REGION Network 47: Call CM Master Virtual Axis (LER_Interlock Summary)
   RUNG wire#powerrail
      #instCmMasterAxisControlInterlockSummary(enableManualCmds := wire#w1, interlockSource := "Unit1.Em3.ControlNodes".cm.Interlock.masterVirtualAxis.source, moduleInterface := "Unit1.Em3.HmiInterface".cmMasterVirtualAxis, controlNode := "Unit1.Em3.ControlNodes".cmMasterVirtualAxis, interlockcGeneral => "Unit1.Em3.ControlNodes".cm.Interlock.masterVirtualAxis.permit.general)
   END_RUNG
   RUNG wire#powerrail
      I_Contact( #statUnitStatus.mode.production )
      Contact( "Unit1.Em3.HmiInterface".webGuid.sequence.monitoring.inStepIdle )
   END_RUNG wire#w1
   // the same network as SCL:
   #instCmMasterAxisControlInterlockSummary(enableManualCmds := NOT #statUnitStatus.mode.production AND "Unit1.Em3.HmiInterface".webGuid.sequence.monitoring.inStepIdle,   // "LER_AxisControl_InterlockSummary"
                           interlockSource := "Unit1.Em3.ControlNodes".cm.Interlock.masterVirtualAxis.source,
                           moduleInterface := "Unit1.Em3.HmiInterface".cmMasterVirtualAxis,
                           controlNode := "Unit1.Em3.ControlNodes".cmMasterVirtualAxis,
                           interlockcGeneral => "Unit1.Em3.ControlNodes".cm.Interlock.masterVirtualAxis.permit.general);
END_REGION

REGION Network 48: Call CM Master Virtual Axis (LBC_AxisControl)
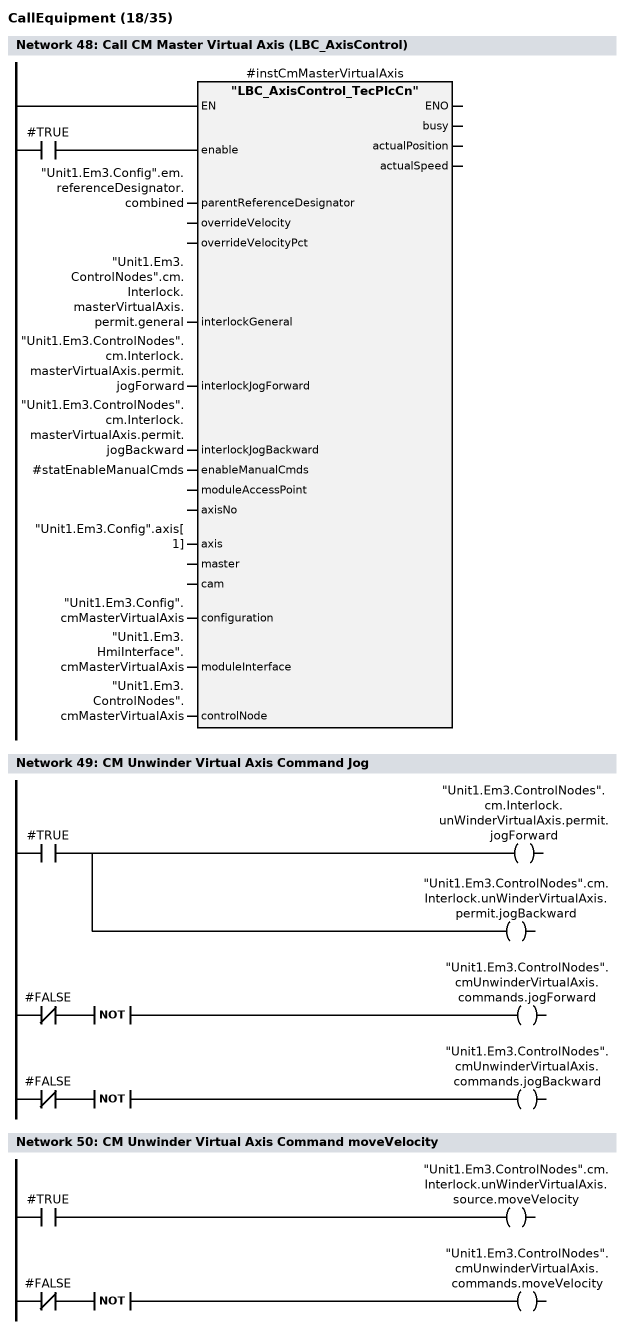
   RUNG wire#powerrail
      #instCmMasterVirtualAxis(enable := wire#w1, parentReferenceDesignator := "Unit1.Em3.Config".em.referenceDesignator.combined, overrideVelocity :=, overrideVelocityPct :=, interlockGeneral := "Unit1.Em3.ControlNodes".cm.Interlock.masterVirtualAxis.permit.general, interlockJogForward := "Unit1.Em3.ControlNodes".cm.Interlock.masterVirtualAxis.permit.jogForward, interlockJogBackward := "Unit1.Em3.ControlNodes".cm.Interlock.masterVirtualAxis.permit.jogBackward, enableManualCmds := #statEnableManualCmds, moduleAccessPoint :=, axisNo :=, axis := "Unit1.Em3.Config".axis[1], master :=, cam :=, configuration := "Unit1.Em3.Config".cmMasterVirtualAxis, moduleInterface := "Unit1.Em3.HmiInterface".cmMasterVirtualAxis, controlNode := "Unit1.Em3.ControlNodes".cmMasterVirtualAxis, busy =>, actualPosition =>, actualSpeed =>)
   END_RUNG
   RUNG wire#powerrail
      Contact( #TRUE )
   END_RUNG wire#w1
   // the same network as SCL:
   #instCmMasterVirtualAxis(enable := #TRUE,   // "LBC_AxisControl_TecPlcCn"
                           parentReferenceDesignator := "Unit1.Em3.Config".em.referenceDesignator.combined,
                           interlockGeneral := "Unit1.Em3.ControlNodes".cm.Interlock.masterVirtualAxis.permit.general,
                           interlockJogForward := "Unit1.Em3.ControlNodes".cm.Interlock.masterVirtualAxis.permit.jogForward,
                           interlockJogBackward := "Unit1.Em3.ControlNodes".cm.Interlock.masterVirtualAxis.permit.jogBackward,
                           enableManualCmds := #statEnableManualCmds,
                           axis := "Unit1.Em3.Config".axis[1],
                           configuration := "Unit1.Em3.Config".cmMasterVirtualAxis,
                           moduleInterface := "Unit1.Em3.HmiInterface".cmMasterVirtualAxis,
                           controlNode := "Unit1.Em3.ControlNodes".cmMasterVirtualAxis);
END_REGION

REGION Network 49: CM Unwinder Virtual Axis Command Jog
   RUNG wire#powerrail
      Contact( #TRUE )
      wire#w1
      Coil( "Unit1.Em3.ControlNodes".cm.Interlock.unWinderVirtualAxis.permit.jogForward )
   END_RUNG
   RUNG wire#w1
      Coil( "Unit1.Em3.ControlNodes".cm.Interlock.unWinderVirtualAxis.permit.jogBackward )
   END_RUNG
   RUNG wire#powerrail
      I_Contact( #FALSE )
      Not()
      Coil( "Unit1.Em3.ControlNodes".cmUnwinderVirtualAxis.commands.jogForward )
   END_RUNG
   RUNG wire#powerrail
      I_Contact( #FALSE )
      Not()
      Coil( "Unit1.Em3.ControlNodes".cmUnwinderVirtualAxis.commands.jogBackward )
   END_RUNG
   // the same network as SCL:
   "Unit1.Em3.ControlNodes".cm.Interlock.unWinderVirtualAxis.permit.jogForward := #TRUE;
   "Unit1.Em3.ControlNodes".cm.Interlock.unWinderVirtualAxis.permit.jogBackward := #TRUE;
   "Unit1.Em3.ControlNodes".cmUnwinderVirtualAxis.commands.jogForward := NOT (NOT #FALSE);
   "Unit1.Em3.ControlNodes".cmUnwinderVirtualAxis.commands.jogBackward := NOT (NOT #FALSE);
END_REGION

REGION Network 50: CM Unwinder Virtual Axis Command moveVelocity
   RUNG wire#powerrail
      Contact( #TRUE )
      Coil( "Unit1.Em3.ControlNodes".cm.Interlock.unWinderVirtualAxis.source.moveVelocity )
   END_RUNG
   RUNG wire#powerrail
      I_Contact( #FALSE )
      Not()
      Coil( "Unit1.Em3.ControlNodes".cmUnwinderVirtualAxis.commands.moveVelocity )
   END_RUNG
   // the same network as SCL:
   "Unit1.Em3.ControlNodes".cm.Interlock.unWinderVirtualAxis.source.moveVelocity := #TRUE;
   "Unit1.Em3.ControlNodes".cmUnwinderVirtualAxis.commands.moveVelocity := NOT (NOT #FALSE);
END_REGION

REGION Network 51: CM Unwinder Virtual Axis Command stop
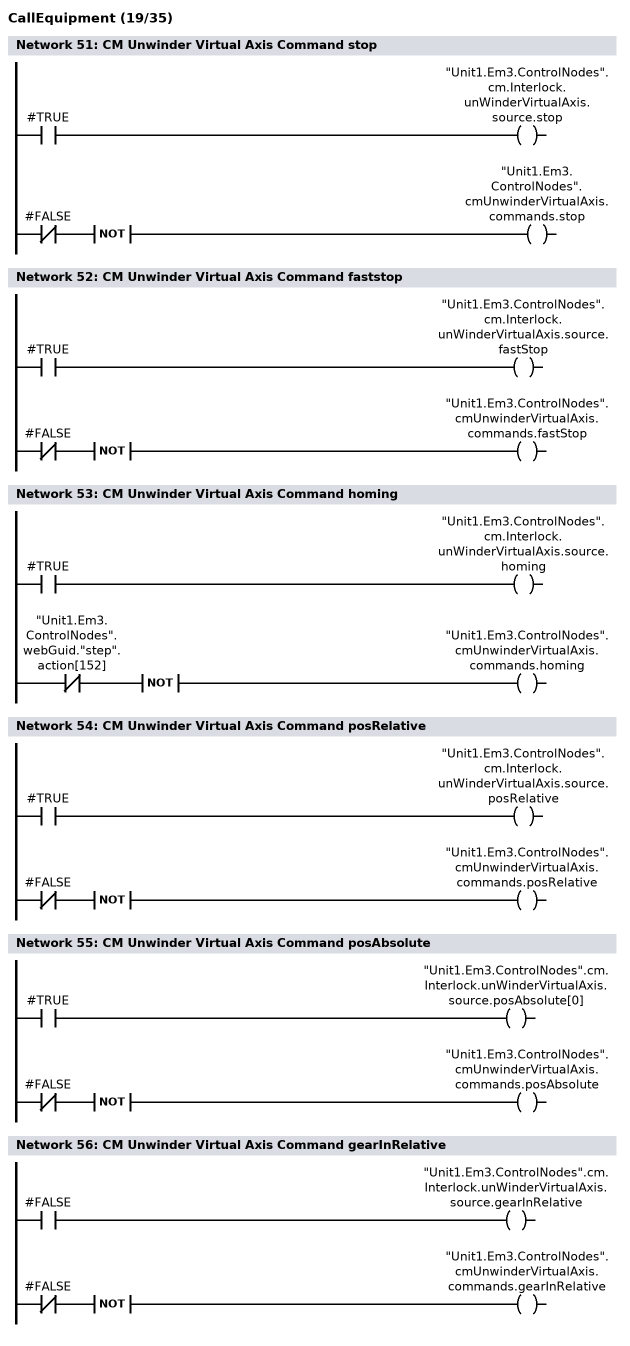
   RUNG wire#powerrail
      Contact( #TRUE )
      Coil( "Unit1.Em3.ControlNodes".cm.Interlock.unWinderVirtualAxis.source.stop )
   END_RUNG
   RUNG wire#powerrail
      I_Contact( #FALSE )
      Not()
      Coil( "Unit1.Em3.ControlNodes".cmUnwinderVirtualAxis.commands.stop )
   END_RUNG
   // the same network as SCL:
   "Unit1.Em3.ControlNodes".cm.Interlock.unWinderVirtualAxis.source.stop := #TRUE;
   "Unit1.Em3.ControlNodes".cmUnwinderVirtualAxis.commands.stop := NOT (NOT #FALSE);
END_REGION

REGION Network 52: CM Unwinder Virtual Axis Command faststop
   RUNG wire#powerrail
      Contact( #TRUE )
      Coil( "Unit1.Em3.ControlNodes".cm.Interlock.unWinderVirtualAxis.source.fastStop )
   END_RUNG
   RUNG wire#powerrail
      I_Contact( #FALSE )
      Not()
      Coil( "Unit1.Em3.ControlNodes".cmUnwinderVirtualAxis.commands.fastStop )
   END_RUNG
   // the same network as SCL:
   "Unit1.Em3.ControlNodes".cm.Interlock.unWinderVirtualAxis.source.fastStop := #TRUE;
   "Unit1.Em3.ControlNodes".cmUnwinderVirtualAxis.commands.fastStop := NOT (NOT #FALSE);
END_REGION

REGION Network 53: CM Unwinder Virtual Axis Command homing
   RUNG wire#powerrail
      Contact( #TRUE )
      Coil( "Unit1.Em3.ControlNodes".cm.Interlock.unWinderVirtualAxis.source.homing )
   END_RUNG
   RUNG wire#powerrail
      I_Contact( "Unit1.Em3.ControlNodes".webGuid."step".action[152] )
      Not()
      Coil( "Unit1.Em3.ControlNodes".cmUnwinderVirtualAxis.commands.homing )
   END_RUNG
   // the same network as SCL:
   "Unit1.Em3.ControlNodes".cm.Interlock.unWinderVirtualAxis.source.homing := #TRUE;
   "Unit1.Em3.ControlNodes".cmUnwinderVirtualAxis.commands.homing := NOT (NOT "Unit1.Em3.ControlNodes".webGuid."step".action[152]);
END_REGION

REGION Network 54: CM Unwinder Virtual Axis Command posRelative
   RUNG wire#powerrail
      Contact( #TRUE )
      Coil( "Unit1.Em3.ControlNodes".cm.Interlock.unWinderVirtualAxis.source.posRelative )
   END_RUNG
   RUNG wire#powerrail
      I_Contact( #FALSE )
      Not()
      Coil( "Unit1.Em3.ControlNodes".cmUnwinderVirtualAxis.commands.posRelative )
   END_RUNG
   // the same network as SCL:
   "Unit1.Em3.ControlNodes".cm.Interlock.unWinderVirtualAxis.source.posRelative := #TRUE;
   "Unit1.Em3.ControlNodes".cmUnwinderVirtualAxis.commands.posRelative := NOT (NOT #FALSE);
END_REGION

REGION Network 55: CM Unwinder Virtual Axis Command posAbsolute
   RUNG wire#powerrail
      Contact( #TRUE )
      Coil( "Unit1.Em3.ControlNodes".cm.Interlock.unWinderVirtualAxis.source.posAbsolute[0] )
   END_RUNG
   RUNG wire#powerrail
      I_Contact( #FALSE )
      Not()
      Coil( "Unit1.Em3.ControlNodes".cmUnwinderVirtualAxis.commands.posAbsolute )
   END_RUNG
   // the same network as SCL:
   "Unit1.Em3.ControlNodes".cm.Interlock.unWinderVirtualAxis.source.posAbsolute[0] := #TRUE;
   "Unit1.Em3.ControlNodes".cmUnwinderVirtualAxis.commands.posAbsolute := NOT (NOT #FALSE);
END_REGION

REGION Network 56: CM Unwinder Virtual Axis Command gearInRelative
   RUNG wire#powerrail
      Contact( #FALSE )
      Coil( "Unit1.Em3.ControlNodes".cm.Interlock.unWinderVirtualAxis.source.gearInRelative )
   END_RUNG
   RUNG wire#powerrail
      I_Contact( #FALSE )
      Not()
      Coil( "Unit1.Em3.ControlNodes".cmUnwinderVirtualAxis.commands.gearInRelative )
   END_RUNG
   // the same network as SCL:
   "Unit1.Em3.ControlNodes".cm.Interlock.unWinderVirtualAxis.source.gearInRelative := #FALSE;
   "Unit1.Em3.ControlNodes".cmUnwinderVirtualAxis.commands.gearInRelative := NOT (NOT #FALSE);
END_REGION

REGION Network 57: CM Unwinder Virtual Axis Command gearInAbsolute
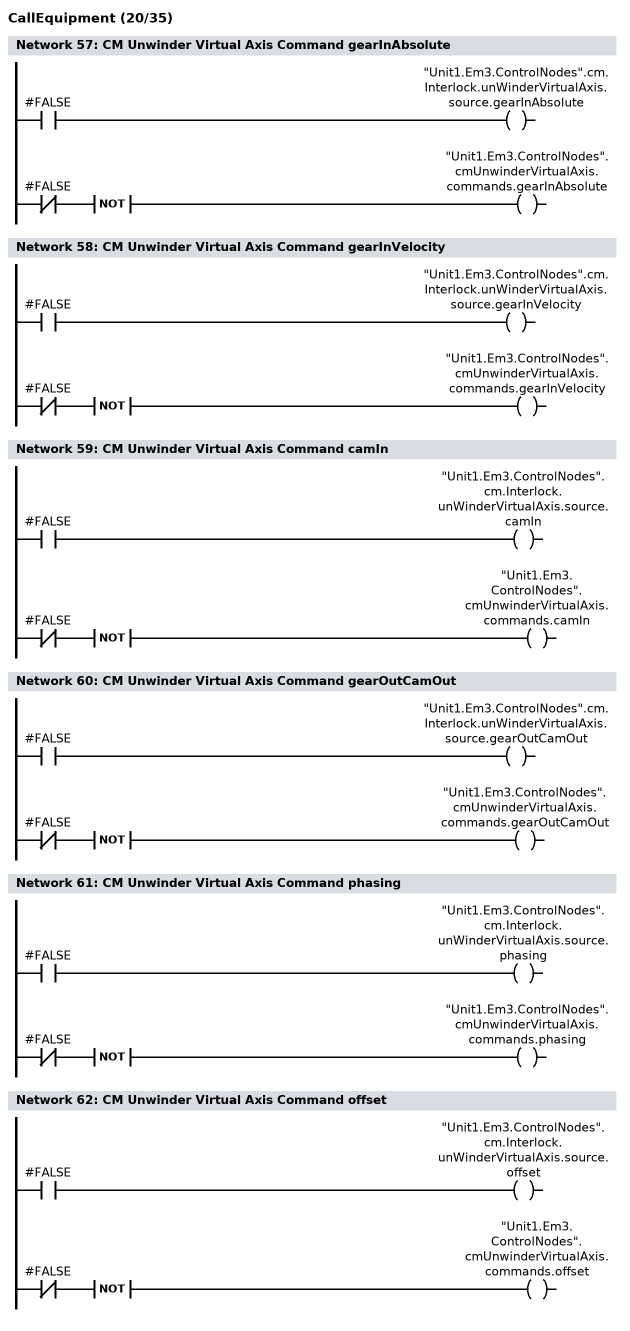
   RUNG wire#powerrail
      Contact( #FALSE )
      Coil( "Unit1.Em3.ControlNodes".cm.Interlock.unWinderVirtualAxis.source.gearInAbsolute )
   END_RUNG
   RUNG wire#powerrail
      I_Contact( #FALSE )
      Not()
      Coil( "Unit1.Em3.ControlNodes".cmUnwinderVirtualAxis.commands.gearInAbsolute )
   END_RUNG
   // the same network as SCL:
   "Unit1.Em3.ControlNodes".cm.Interlock.unWinderVirtualAxis.source.gearInAbsolute := #FALSE;
   "Unit1.Em3.ControlNodes".cmUnwinderVirtualAxis.commands.gearInAbsolute := NOT (NOT #FALSE);
END_REGION

REGION Network 58: CM Unwinder Virtual Axis Command gearInVelocity
   RUNG wire#powerrail
      Contact( #FALSE )
      Coil( "Unit1.Em3.ControlNodes".cm.Interlock.unWinderVirtualAxis.source.gearInVelocity )
   END_RUNG
   RUNG wire#powerrail
      I_Contact( #FALSE )
      Not()
      Coil( "Unit1.Em3.ControlNodes".cmUnwinderVirtualAxis.commands.gearInVelocity )
   END_RUNG
   // the same network as SCL:
   "Unit1.Em3.ControlNodes".cm.Interlock.unWinderVirtualAxis.source.gearInVelocity := #FALSE;
   "Unit1.Em3.ControlNodes".cmUnwinderVirtualAxis.commands.gearInVelocity := NOT (NOT #FALSE);
END_REGION

REGION Network 59: CM Unwinder Virtual Axis Command camIn
   RUNG wire#powerrail
      Contact( #FALSE )
      Coil( "Unit1.Em3.ControlNodes".cm.Interlock.unWinderVirtualAxis.source.camIn )
   END_RUNG
   RUNG wire#powerrail
      I_Contact( #FALSE )
      Not()
      Coil( "Unit1.Em3.ControlNodes".cmUnwinderVirtualAxis.commands.camIn )
   END_RUNG
   // the same network as SCL:
   "Unit1.Em3.ControlNodes".cm.Interlock.unWinderVirtualAxis.source.camIn := #FALSE;
   "Unit1.Em3.ControlNodes".cmUnwinderVirtualAxis.commands.camIn := NOT (NOT #FALSE);
END_REGION

REGION Network 60: CM Unwinder Virtual Axis Command gearOutCamOut
   RUNG wire#powerrail
      Contact( #FALSE )
      Coil( "Unit1.Em3.ControlNodes".cm.Interlock.unWinderVirtualAxis.source.gearOutCamOut )
   END_RUNG
   RUNG wire#powerrail
      I_Contact( #FALSE )
      Not()
      Coil( "Unit1.Em3.ControlNodes".cmUnwinderVirtualAxis.commands.gearOutCamOut )
   END_RUNG
   // the same network as SCL:
   "Unit1.Em3.ControlNodes".cm.Interlock.unWinderVirtualAxis.source.gearOutCamOut := #FALSE;
   "Unit1.Em3.ControlNodes".cmUnwinderVirtualAxis.commands.gearOutCamOut := NOT (NOT #FALSE);
END_REGION

REGION Network 61: CM Unwinder Virtual Axis Command phasing
   RUNG wire#powerrail
      Contact( #FALSE )
      Coil( "Unit1.Em3.ControlNodes".cm.Interlock.unWinderVirtualAxis.source.phasing )
   END_RUNG
   RUNG wire#powerrail
      I_Contact( #FALSE )
      Not()
      Coil( "Unit1.Em3.ControlNodes".cmUnwinderVirtualAxis.commands.phasing )
   END_RUNG
   // the same network as SCL:
   "Unit1.Em3.ControlNodes".cm.Interlock.unWinderVirtualAxis.source.phasing := #FALSE;
   "Unit1.Em3.ControlNodes".cmUnwinderVirtualAxis.commands.phasing := NOT (NOT #FALSE);
END_REGION

REGION Network 62: CM Unwinder Virtual Axis Command offset
   RUNG wire#powerrail
      Contact( #FALSE )
      Coil( "Unit1.Em3.ControlNodes".cm.Interlock.unWinderVirtualAxis.source.offset )
   END_RUNG
   RUNG wire#powerrail
      I_Contact( #FALSE )
      Not()
      Coil( "Unit1.Em3.ControlNodes".cmUnwinderVirtualAxis.commands.offset )
   END_RUNG
   // the same network as SCL:
   "Unit1.Em3.ControlNodes".cm.Interlock.unWinderVirtualAxis.source.offset := #FALSE;
   "Unit1.Em3.ControlNodes".cmUnwinderVirtualAxis.commands.offset := NOT (NOT #FALSE);
END_REGION

REGION Network 63: Call CM Unwinder Virtual Axis (LER_Interlock Summary)
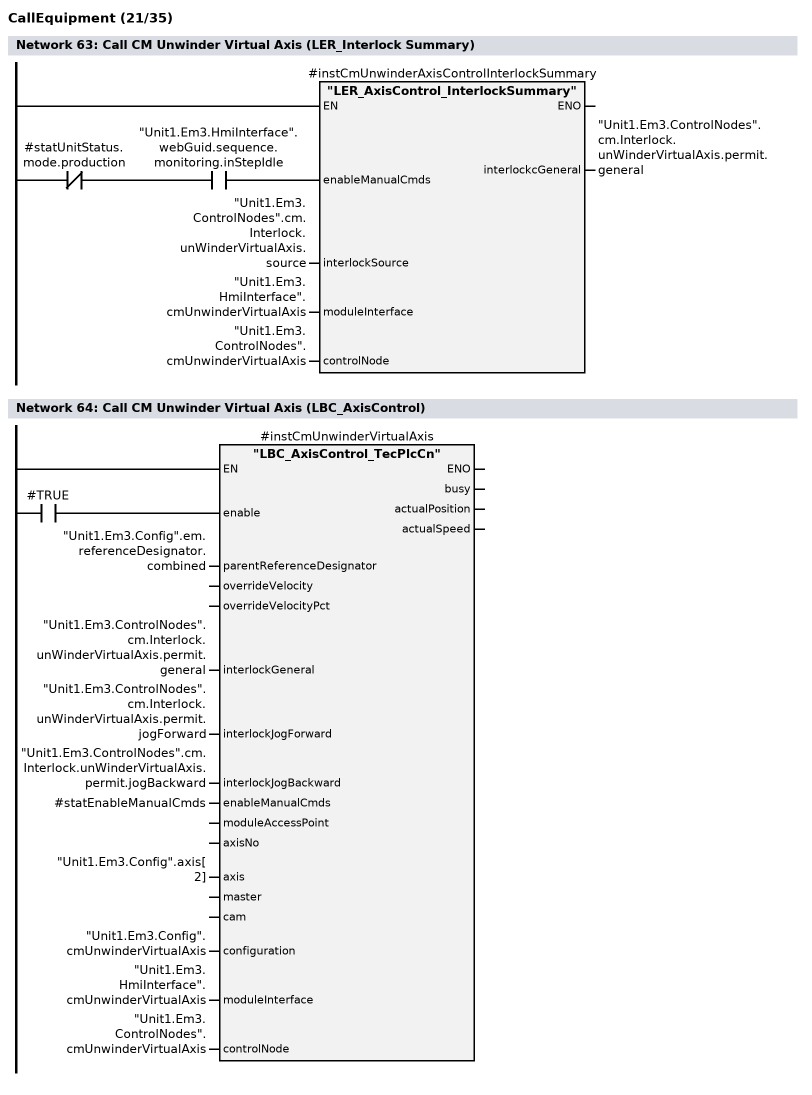
   RUNG wire#powerrail
      #instCmUnwinderAxisControlInterlockSummary(enableManualCmds := wire#w1, interlockSource := "Unit1.Em3.ControlNodes".cm.Interlock.unWinderVirtualAxis.source, moduleInterface := "Unit1.Em3.HmiInterface".cmUnwinderVirtualAxis, controlNode := "Unit1.Em3.ControlNodes".cmUnwinderVirtualAxis, interlockcGeneral => "Unit1.Em3.ControlNodes".cm.Interlock.unWinderVirtualAxis.permit.general)
   END_RUNG
   RUNG wire#powerrail
      I_Contact( #statUnitStatus.mode.production )
      Contact( "Unit1.Em3.HmiInterface".webGuid.sequence.monitoring.inStepIdle )
   END_RUNG wire#w1
   // the same network as SCL:
   #instCmUnwinderAxisControlInterlockSummary(enableManualCmds := NOT #statUnitStatus.mode.production AND "Unit1.Em3.HmiInterface".webGuid.sequence.monitoring.inStepIdle,   // "LER_AxisControl_InterlockSummary"
                           interlockSource := "Unit1.Em3.ControlNodes".cm.Interlock.unWinderVirtualAxis.source,
                           moduleInterface := "Unit1.Em3.HmiInterface".cmUnwinderVirtualAxis,
                           controlNode := "Unit1.Em3.ControlNodes".cmUnwinderVirtualAxis,
                           interlockcGeneral => "Unit1.Em3.ControlNodes".cm.Interlock.unWinderVirtualAxis.permit.general);
END_REGION

REGION Network 64: Call CM Unwinder Virtual Axis (LBC_AxisControl)
   RUNG wire#powerrail
      #instCmUnwinderVirtualAxis(enable := wire#w1, parentReferenceDesignator := "Unit1.Em3.Config".em.referenceDesignator.combined, overrideVelocity :=, overrideVelocityPct :=, interlockGeneral := "Unit1.Em3.ControlNodes".cm.Interlock.unWinderVirtualAxis.permit.general, interlockJogForward := "Unit1.Em3.ControlNodes".cm.Interlock.unWinderVirtualAxis.permit.jogForward, interlockJogBackward := "Unit1.Em3.ControlNodes".cm.Interlock.unWinderVirtualAxis.permit.jogBackward, enableManualCmds := #statEnableManualCmds, moduleAccessPoint :=, axisNo :=, axis := "Unit1.Em3.Config".axis[2], master :=, cam :=, configuration := "Unit1.Em3.Config".cmUnwinderVirtualAxis, moduleInterface := "Unit1.Em3.HmiInterface".cmUnwinderVirtualAxis, controlNode := "Unit1.Em3.ControlNodes".cmUnwinderVirtualAxis, busy =>, actualPosition =>, actualSpeed =>)
   END_RUNG
   RUNG wire#powerrail
      Contact( #TRUE )
   END_RUNG wire#w1
   // the same network as SCL:
   #instCmUnwinderVirtualAxis(enable := #TRUE,   // "LBC_AxisControl_TecPlcCn"
                           parentReferenceDesignator := "Unit1.Em3.Config".em.referenceDesignator.combined,
                           interlockGeneral := "Unit1.Em3.ControlNodes".cm.Interlock.unWinderVirtualAxis.permit.general,
                           interlockJogForward := "Unit1.Em3.ControlNodes".cm.Interlock.unWinderVirtualAxis.permit.jogForward,
                           interlockJogBackward := "Unit1.Em3.ControlNodes".cm.Interlock.unWinderVirtualAxis.permit.jogBackward,
                           enableManualCmds := #statEnableManualCmds,
                           axis := "Unit1.Em3.Config".axis[2],
                           configuration := "Unit1.Em3.Config".cmUnwinderVirtualAxis,
                           moduleInterface := "Unit1.Em3.HmiInterface".cmUnwinderVirtualAxis,
                           controlNode := "Unit1.Em3.ControlNodes".cmUnwinderVirtualAxis);
END_REGION

REGION Network 65: ******************** Control Modules (TwoWayActuator) ********************
   // Call control modules that are actuators after the em logic (jobs and sequence), so that the latest commands are applied to the actuators.
END_REGION

REGION Network 66: Reset CMS
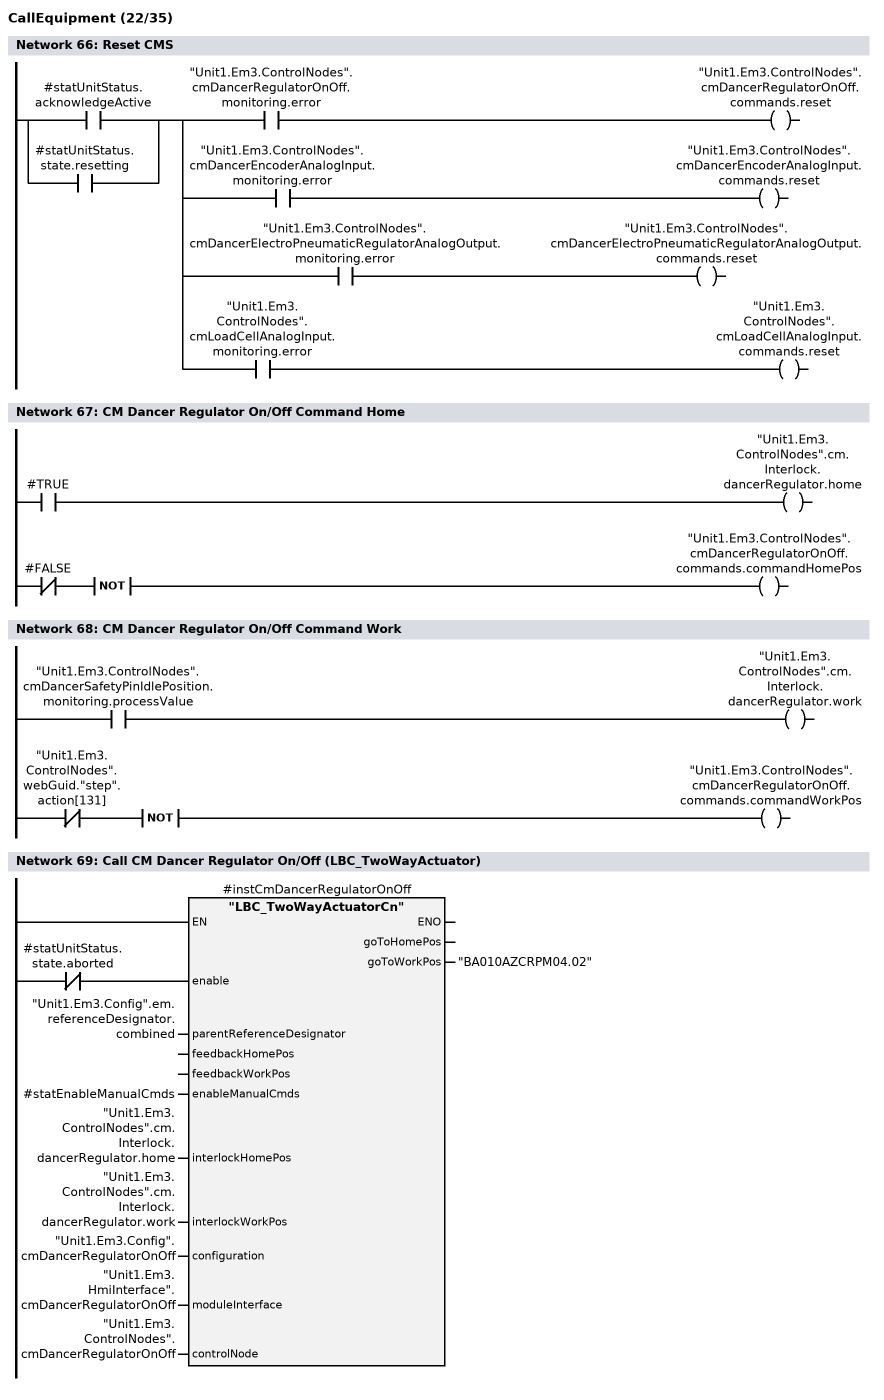
   RUNG wire#powerrail
      Contact( #statUnitStatus.acknowledgeActive )
      wire#w1
      Contact( "Unit1.Em3.ControlNodes".cmDancerRegulatorOnOff.monitoring.error )
      Coil( "Unit1.Em3.ControlNodes".cmDancerRegulatorOnOff.commands.reset )
   END_RUNG
   RUNG wire#powerrail
      Contact( #statUnitStatus.state.resetting )
   END_RUNG wire#w1
   RUNG wire#w1
      Contact( "Unit1.Em3.ControlNodes".cmDancerEncoderAnalogInput.monitoring.error )
      Coil( "Unit1.Em3.ControlNodes".cmDancerEncoderAnalogInput.commands.reset )
   END_RUNG
   RUNG wire#w1
      Contact( "Unit1.Em3.ControlNodes".cmDancerElectroPneumaticRegulatorAnalogOutput.monitoring.error )
      Coil( "Unit1.Em3.ControlNodes".cmDancerElectroPneumaticRegulatorAnalogOutput.commands.reset )
   END_RUNG
   RUNG wire#w1
      Contact( "Unit1.Em3.ControlNodes".cmLoadCellAnalogInput.monitoring.error )
      Coil( "Unit1.Em3.ControlNodes".cmLoadCellAnalogInput.commands.reset )
   END_RUNG
   // the same network as SCL:
   #_w1 := #statUnitStatus.acknowledgeActive OR #statUnitStatus.state.resetting;
   "Unit1.Em3.ControlNodes".cmDancerRegulatorOnOff.commands.reset := #_w1 AND "Unit1.Em3.ControlNodes".cmDancerRegulatorOnOff.monitoring.error;
   "Unit1.Em3.ControlNodes".cmDancerEncoderAnalogInput.commands.reset := #_w1 AND "Unit1.Em3.ControlNodes".cmDancerEncoderAnalogInput.monitoring.error;
   "Unit1.Em3.ControlNodes".cmDancerElectroPneumaticRegulatorAnalogOutput.commands.reset := #_w1 AND "Unit1.Em3.ControlNodes".cmDancerElectroPneumaticRegulatorAnalogOutput.monitoring.error;
   "Unit1.Em3.ControlNodes".cmLoadCellAnalogInput.commands.reset := #_w1 AND "Unit1.Em3.ControlNodes".cmLoadCellAnalogInput.monitoring.error;
END_REGION

REGION Network 67: CM Dancer Regulator On/Off Command Home
   RUNG wire#powerrail
      Contact( #TRUE )
      Coil( "Unit1.Em3.ControlNodes".cm.Interlock.dancerRegulator.home )
   END_RUNG
   RUNG wire#powerrail
      I_Contact( #FALSE )
      Not()
      Coil( "Unit1.Em3.ControlNodes".cmDancerRegulatorOnOff.commands.commandHomePos )
   END_RUNG
   // the same network as SCL:
   "Unit1.Em3.ControlNodes".cm.Interlock.dancerRegulator.home := #TRUE;
   "Unit1.Em3.ControlNodes".cmDancerRegulatorOnOff.commands.commandHomePos := NOT (NOT #FALSE);
END_REGION

REGION Network 68: CM Dancer Regulator On/Off Command Work
   RUNG wire#powerrail
      Contact( "Unit1.Em3.ControlNodes".cmDancerSafetyPinIdlePosition.monitoring.processValue )
      Coil( "Unit1.Em3.ControlNodes".cm.Interlock.dancerRegulator.work )
   END_RUNG
   RUNG wire#powerrail
      I_Contact( "Unit1.Em3.ControlNodes".webGuid."step".action[131] )
      Not()
      Coil( "Unit1.Em3.ControlNodes".cmDancerRegulatorOnOff.commands.commandWorkPos )
   END_RUNG
   // the same network as SCL:
   "Unit1.Em3.ControlNodes".cm.Interlock.dancerRegulator.work := "Unit1.Em3.ControlNodes".cmDancerSafetyPinIdlePosition.monitoring.processValue;
   "Unit1.Em3.ControlNodes".cmDancerRegulatorOnOff.commands.commandWorkPos := NOT (NOT "Unit1.Em3.ControlNodes".webGuid."step".action[131]);
END_REGION

REGION Network 69: Call CM Dancer Regulator On/Off (LBC_TwoWayActuator)
   RUNG wire#powerrail
      #instCmDancerRegulatorOnOff(enable := wire#w1, parentReferenceDesignator := "Unit1.Em3.Config".em.referenceDesignator.combined, feedbackHomePos :=, feedbackWorkPos :=, enableManualCmds := #statEnableManualCmds, interlockHomePos := "Unit1.Em3.ControlNodes".cm.Interlock.dancerRegulator.home, interlockWorkPos := "Unit1.Em3.ControlNodes".cm.Interlock.dancerRegulator.work, configuration := "Unit1.Em3.Config".cmDancerRegulatorOnOff, moduleInterface := "Unit1.Em3.HmiInterface".cmDancerRegulatorOnOff, controlNode := "Unit1.Em3.ControlNodes".cmDancerRegulatorOnOff, goToHomePos =>, goToWorkPos => "BA010AZCRPM04.02")
   END_RUNG
   RUNG wire#powerrail
      I_Contact( #statUnitStatus.state.aborted )
   END_RUNG wire#w1
   // the same network as SCL:
   #instCmDancerRegulatorOnOff(enable := NOT #statUnitStatus.state.aborted,   // "LBC_TwoWayActuatorCn"
                           parentReferenceDesignator := "Unit1.Em3.Config".em.referenceDesignator.combined,
                           enableManualCmds := #statEnableManualCmds,
                           interlockHomePos := "Unit1.Em3.ControlNodes".cm.Interlock.dancerRegulator.home,
                           interlockWorkPos := "Unit1.Em3.ControlNodes".cm.Interlock.dancerRegulator.work,
                           configuration := "Unit1.Em3.Config".cmDancerRegulatorOnOff,
                           moduleInterface := "Unit1.Em3.HmiInterface".cmDancerRegulatorOnOff,
                           controlNode := "Unit1.Em3.ControlNodes".cmDancerRegulatorOnOff,
                           goToWorkPos => "BA010AZCRPM04.02");
END_REGION

REGION Network 70: ******************** Control Modules (Accessories) ********************
   // Call control modules that are actuators after the em logic (jobs and sequence), so that the latest commands are applied to the actuators.
END_REGION

REGION Network 71: Reset CMS
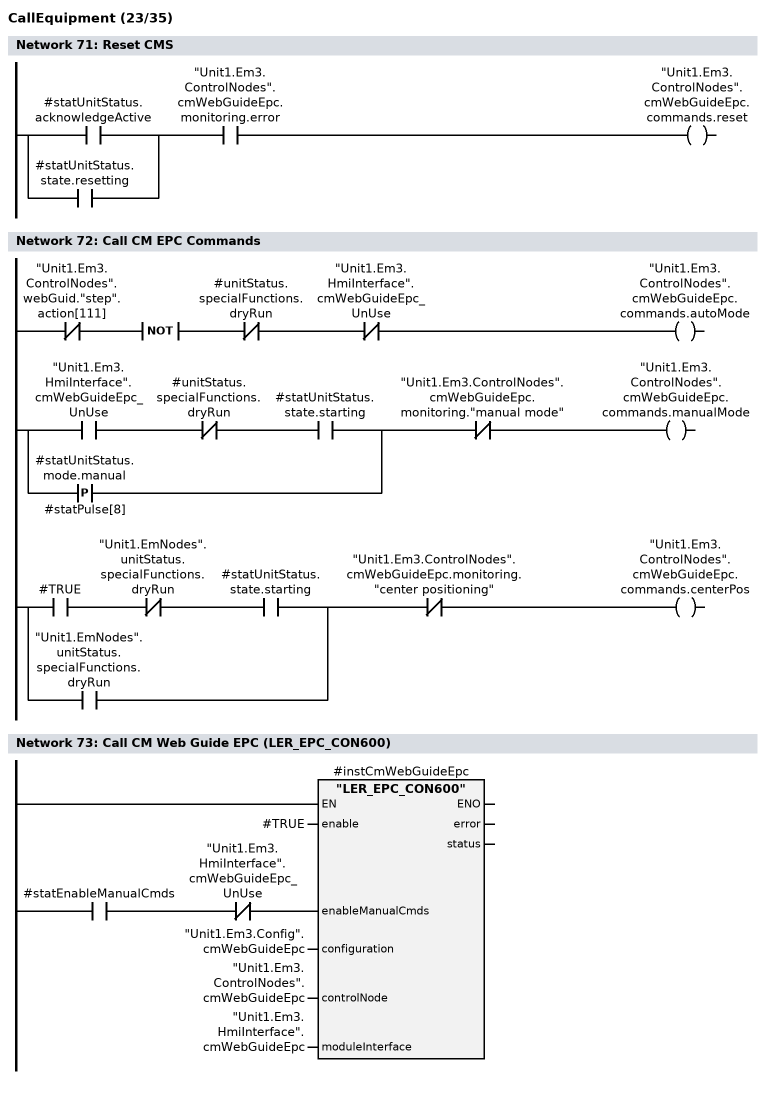
   RUNG wire#powerrail
      Contact( #statUnitStatus.acknowledgeActive )
      wire#w1
      Contact( "Unit1.Em3.ControlNodes".cmWebGuideEpc.monitoring.error )
      Coil( "Unit1.Em3.ControlNodes".cmWebGuideEpc.commands.reset )
   END_RUNG
   RUNG wire#powerrail
      Contact( #statUnitStatus.state.resetting )
   END_RUNG wire#w1
   // the same network as SCL:
   "Unit1.Em3.ControlNodes".cmWebGuideEpc.commands.reset := (#statUnitStatus.acknowledgeActive OR #statUnitStatus.state.resetting) AND "Unit1.Em3.ControlNodes".cmWebGuideEpc.monitoring.error;
END_REGION

REGION Network 72: Call CM EPC Commands
   RUNG wire#powerrail
      I_Contact( "Unit1.Em3.ControlNodes".webGuid."step".action[111] )
      Not()
      I_Contact( #unitStatus.specialFunctions.dryRun )
      I_Contact( "Unit1.Em3.HmiInterface".cmWebGuideEpc_UnUse )
      Coil( "Unit1.Em3.ControlNodes".cmWebGuideEpc.commands.autoMode )
   END_RUNG
   RUNG wire#powerrail
      Contact( "Unit1.Em3.HmiInterface".cmWebGuideEpc_UnUse )
      I_Contact( #unitStatus.specialFunctions.dryRun )
      Contact( #statUnitStatus.state.starting )
      wire#w1
      I_Contact( "Unit1.Em3.ControlNodes".cmWebGuideEpc.monitoring."manual mode" )
      Coil( "Unit1.Em3.ControlNodes".cmWebGuideEpc.commands.manualMode )
   END_RUNG
   RUNG wire#powerrail
      P_Contact(operand := #statUnitStatus.mode.manual, bit := #statPulse[8])
   END_RUNG wire#w1
   RUNG wire#powerrail
      Contact( #TRUE )
      I_Contact( "Unit1.EmNodes".unitStatus.specialFunctions.dryRun )
      Contact( #statUnitStatus.state.starting )
      wire#w2
      I_Contact( "Unit1.Em3.ControlNodes".cmWebGuideEpc.monitoring."center positioning" )
      Coil( "Unit1.Em3.ControlNodes".cmWebGuideEpc.commands.centerPos )
   END_RUNG
   RUNG wire#powerrail
      Contact( "Unit1.EmNodes".unitStatus.specialFunctions.dryRun )
   END_RUNG wire#w2
   // the same network as SCL:
   "Unit1.Em3.ControlNodes".cmWebGuideEpc.commands.autoMode := NOT (NOT "Unit1.Em3.ControlNodes".webGuid."step".action[111]) AND NOT #unitStatus.specialFunctions.dryRun AND NOT "Unit1.Em3.HmiInterface".cmWebGuideEpc_UnUse;
   #_w1 := #statUnitStatus.mode.manual AND NOT #statPulse[8];   // rising edge of #statUnitStatus.mode.manual
   #statPulse[8] := #statUnitStatus.mode.manual;
   "Unit1.Em3.ControlNodes".cmWebGuideEpc.commands.manualMode := (("Unit1.Em3.HmiInterface".cmWebGuideEpc_UnUse AND NOT #unitStatus.specialFunctions.dryRun AND #statUnitStatus.state.starting) OR #_w1) AND NOT "Unit1.Em3.ControlNodes".cmWebGuideEpc.monitoring."manual mode";
   "Unit1.Em3.ControlNodes".cmWebGuideEpc.commands.centerPos := ((#TRUE AND NOT "Unit1.EmNodes".unitStatus.specialFunctions.dryRun AND #statUnitStatus.state.starting) OR "Unit1.EmNodes".unitStatus.specialFunctions.dryRun) AND NOT "Unit1.Em3.ControlNodes".cmWebGuideEpc.monitoring."center positioning";
END_REGION

REGION Network 73: Call CM Web Guide EPC (LER_EPC_CON600)
   RUNG wire#powerrail
      #instCmWebGuideEpc(enableManualCmds := wire#w1, enable := #TRUE, configuration := "Unit1.Em3.Config".cmWebGuideEpc, controlNode := "Unit1.Em3.ControlNodes".cmWebGuideEpc, moduleInterface := "Unit1.Em3.HmiInterface".cmWebGuideEpc, error =>, status =>)
   END_RUNG
   RUNG wire#powerrail
      Contact( #statEnableManualCmds )
      I_Contact( "Unit1.Em3.HmiInterface".cmWebGuideEpc_UnUse )
   END_RUNG wire#w1
   // the same network as SCL:
   #instCmWebGuideEpc(enable := #TRUE,   // "LER_EPC_CON600"
                      enableManualCmds := #statEnableManualCmds AND NOT "Unit1.Em3.HmiInterface".cmWebGuideEpc_UnUse,
                      configuration := "Unit1.Em3.Config".cmWebGuideEpc,
                      controlNode := "Unit1.Em3.ControlNodes".cmWebGuideEpc,
                      moduleInterface := "Unit1.Em3.HmiInterface".cmWebGuideEpc);
END_REGION

REGION Network 74: ******************** Motion Interface (SyncMotion) ********************
END_REGION

REGION Network 75: Call LER_CheckCamRecipeChanged
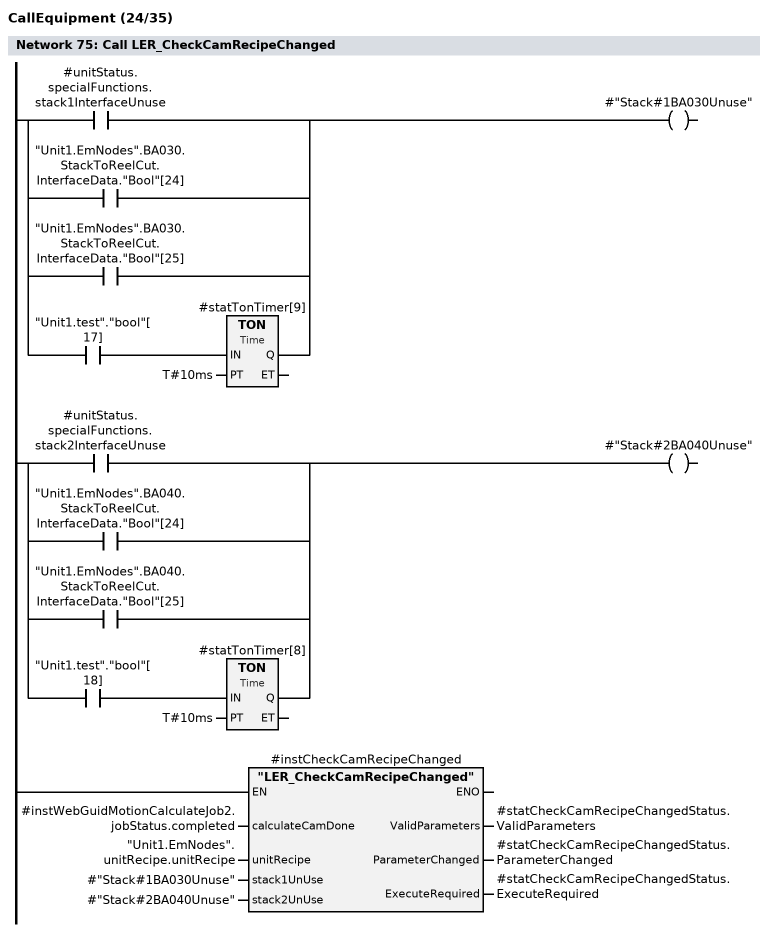
   RUNG wire#powerrail
      Contact( #unitStatus.specialFunctions.stack1InterfaceUnuse )
      wire#w1
      Coil( #"Stack#1BA030Unuse" )
   END_RUNG
   RUNG wire#powerrail
      Contact( "Unit1.EmNodes".BA030.StackToReelCut.InterfaceData."Bool"[24] )
   END_RUNG wire#w1
   RUNG wire#powerrail
      Contact( "Unit1.EmNodes".BA030.StackToReelCut.InterfaceData."Bool"[25] )
   END_RUNG wire#w1
   RUNG wire#powerrail
      Contact( "Unit1.test"."bool"[17] )
      { S7_Templates := "time_type := Time" } #statTonTimer[9].TON(pt := T#10ms, et =>)
   END_RUNG wire#w1
   RUNG wire#powerrail
      Contact( #unitStatus.specialFunctions.stack2InterfaceUnuse )
      wire#w2
      Coil( #"Stack#2BA040Unuse" )
   END_RUNG
   RUNG wire#powerrail
      Contact( "Unit1.EmNodes".BA040.StackToReelCut.InterfaceData."Bool"[24] )
   END_RUNG wire#w2
   RUNG wire#powerrail
      Contact( "Unit1.EmNodes".BA040.StackToReelCut.InterfaceData."Bool"[25] )
   END_RUNG wire#w2
   RUNG wire#powerrail
      Contact( "Unit1.test"."bool"[18] )
      { S7_Templates := "time_type := Time" } #statTonTimer[8].TON(pt := T#10ms, et =>)
   END_RUNG wire#w2
   RUNG wire#powerrail
      #instCheckCamRecipeChanged(calculateCamDone := #instWebGuidMotionCalculateJob2.jobStatus.completed, unitRecipe := "Unit1.EmNodes".unitRecipe.unitRecipe, stack1UnUse := #"Stack#1BA030Unuse", stack2UnUse := #"Stack#2BA040Unuse", ValidParameters => #statCheckCamRecipeChangedStatus.ValidParameters, ParameterChanged => #statCheckCamRecipeChangedStatus.ParameterChanged, ExecuteRequired => #statCheckCamRecipeChangedStatus.ExecuteRequired)
   END_RUNG
   // the same network as SCL:
   #statTonTimer[9].TON(IN := "Unit1.test"."bool"[17], PT := T#10ms);
   #"Stack#1BA030Unuse" := #unitStatus.specialFunctions.stack1InterfaceUnuse OR "Unit1.EmNodes".BA030.StackToReelCut.InterfaceData."Bool"[24] OR "Unit1.EmNodes".BA030.StackToReelCut.InterfaceData."Bool"[25] OR #statTonTimer[9].Q;
   #statTonTimer[8].TON(IN := "Unit1.test"."bool"[18], PT := T#10ms);
   #"Stack#2BA040Unuse" := #unitStatus.specialFunctions.stack2InterfaceUnuse OR "Unit1.EmNodes".BA040.StackToReelCut.InterfaceData."Bool"[24] OR "Unit1.EmNodes".BA040.StackToReelCut.InterfaceData."Bool"[25] OR #statTonTimer[8].Q;
   #instCheckCamRecipeChanged(calculateCamDone := #instWebGuidMotionCalculateJob2.jobStatus.completed,   // "LER_CheckCamRecipeChanged"
                           unitRecipe := "Unit1.EmNodes".unitRecipe.unitRecipe,
                           stack1UnUse := #"Stack#1BA030Unuse",
                           stack2UnUse := #"Stack#2BA040Unuse",
                           ValidParameters => #statCheckCamRecipeChangedStatus.ValidParameters,
                           ParameterChanged => #statCheckCamRecipeChangedStatus.ParameterChanged,
                           ExecuteRequired => #statCheckCamRecipeChangedStatus.ExecuteRequired);
END_REGION

REGION Network 76: Commands Dancer
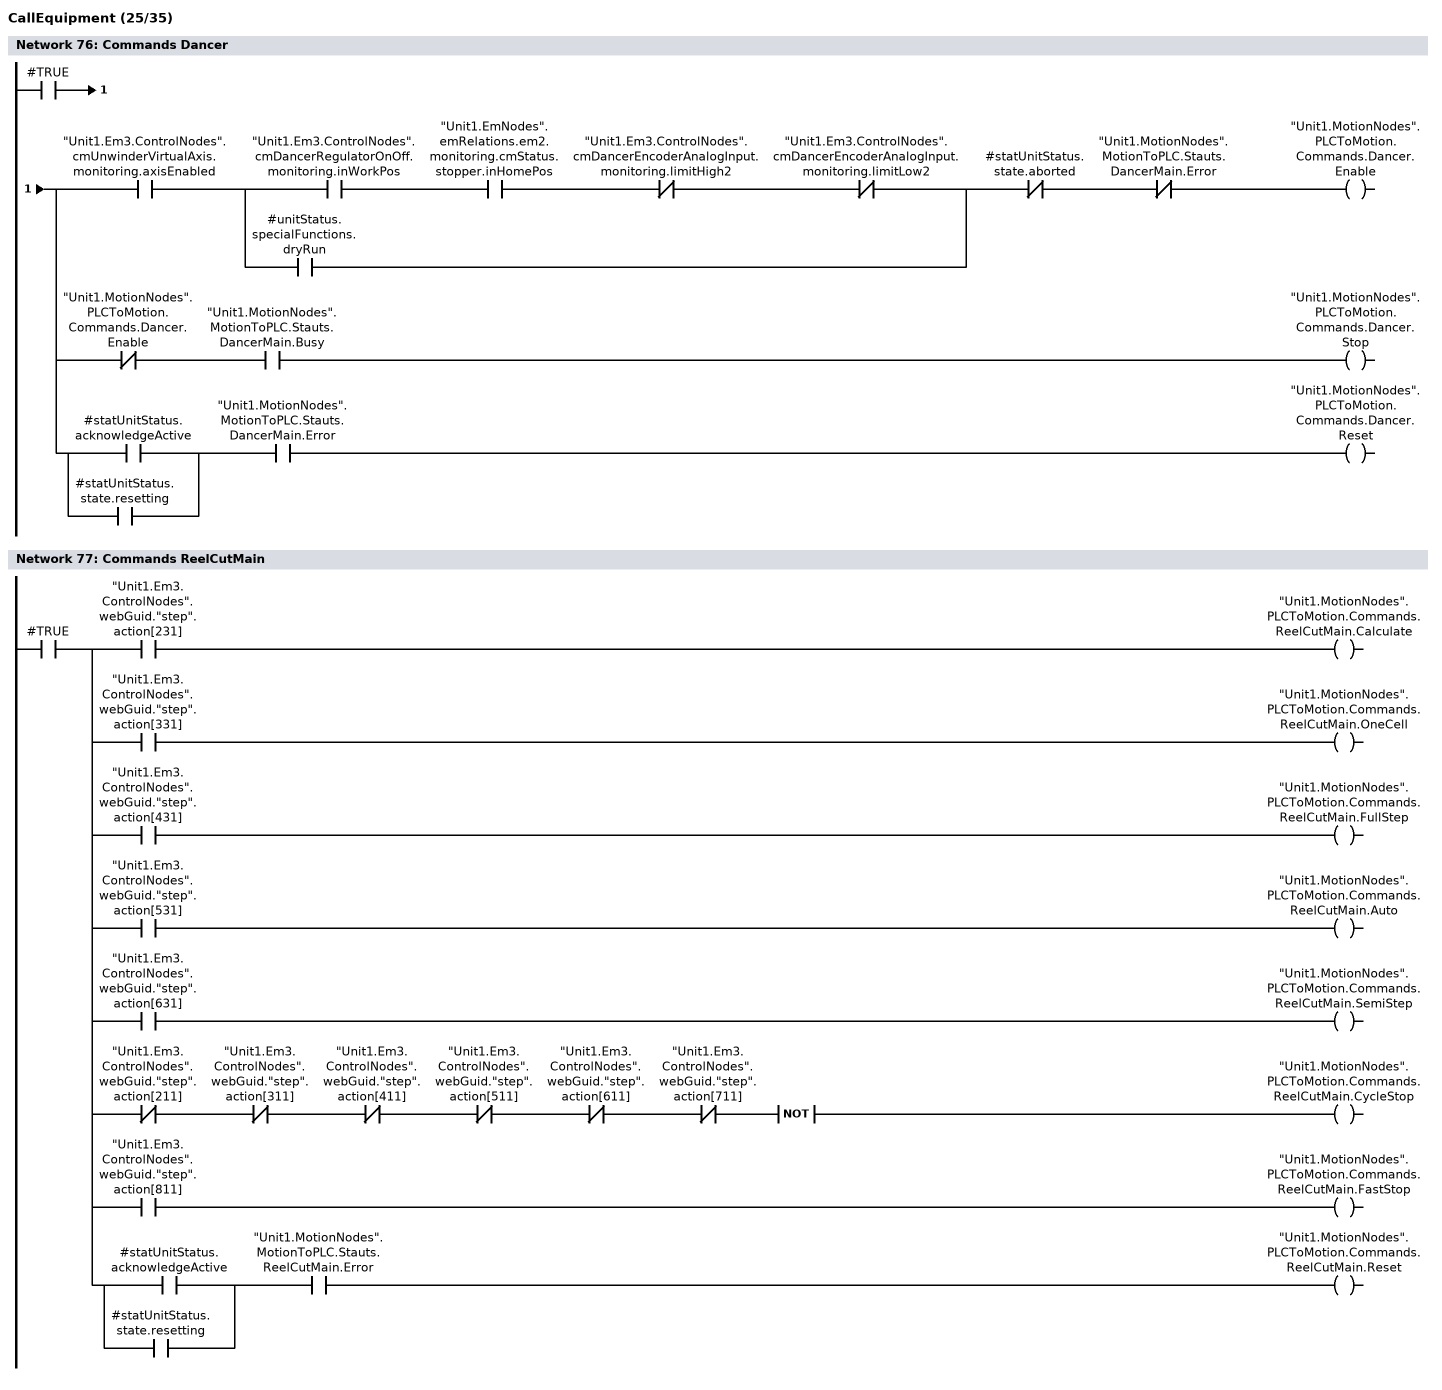
   RUNG wire#powerrail
      Contact( #TRUE )
      wire#w1
      Contact( "Unit1.Em3.ControlNodes".cmUnwinderVirtualAxis.monitoring.axisEnabled )
      wire#w2
      Contact( "Unit1.Em3.ControlNodes".cmDancerRegulatorOnOff.monitoring.inWorkPos )
      Contact( "Unit1.EmNodes".emRelations.em2.monitoring.cmStatus.stopper.inHomePos )
      I_Contact( "Unit1.Em3.ControlNodes".cmDancerEncoderAnalogInput.monitoring.limitHigh2 )
      I_Contact( "Unit1.Em3.ControlNodes".cmDancerEncoderAnalogInput.monitoring.limitLow2 )
      wire#w3
      I_Contact( #statUnitStatus.state.aborted )
      I_Contact( "Unit1.MotionNodes".MotionToPLC.Stauts.DancerMain.Error )
      Coil( "Unit1.MotionNodes".PLCToMotion.Commands.Dancer.Enable )
   END_RUNG
   RUNG wire#w2
      Contact( #unitStatus.specialFunctions.dryRun )
   END_RUNG wire#w3
   RUNG wire#w1
      I_Contact( "Unit1.MotionNodes".PLCToMotion.Commands.Dancer.Enable )
      Contact( "Unit1.MotionNodes".MotionToPLC.Stauts.DancerMain.Busy )
      Coil( "Unit1.MotionNodes".PLCToMotion.Commands.Dancer.Stop )
   END_RUNG
   RUNG wire#w1
      Contact( #statUnitStatus.acknowledgeActive )
      wire#w4
      Contact( "Unit1.MotionNodes".MotionToPLC.Stauts.DancerMain.Error )
      Coil( "Unit1.MotionNodes".PLCToMotion.Commands.Dancer.Reset )
   END_RUNG
   RUNG wire#w1
      Contact( #statUnitStatus.state.resetting )
   END_RUNG wire#w4
   // the same network as SCL:
   "Unit1.MotionNodes".PLCToMotion.Commands.Dancer.Enable := #TRUE AND "Unit1.Em3.ControlNodes".cmUnwinderVirtualAxis.monitoring.axisEnabled AND (("Unit1.Em3.ControlNodes".cmDancerRegulatorOnOff.monitoring.inWorkPos AND "Unit1.EmNodes".emRelations.em2.monitoring.cmStatus.stopper.inHomePos AND NOT "Unit1.Em3.ControlNodes".cmDancerEncoderAnalogInput.monitoring.limitHigh2 AND NOT "Unit1.Em3.ControlNodes".cmDancerEncoderAnalogInput.monitoring.limitLow2) OR #unitStatus.specialFunctions.dryRun) AND NOT #statUnitStatus.state.aborted AND NOT "Unit1.MotionNodes".MotionToPLC.Stauts.DancerMain.Error;
   "Unit1.MotionNodes".PLCToMotion.Commands.Dancer.Stop := #TRUE AND NOT "Unit1.MotionNodes".PLCToMotion.Commands.Dancer.Enable AND "Unit1.MotionNodes".MotionToPLC.Stauts.DancerMain.Busy;
   "Unit1.MotionNodes".PLCToMotion.Commands.Dancer.Reset := #TRUE AND (#statUnitStatus.acknowledgeActive OR #statUnitStatus.state.resetting) AND "Unit1.MotionNodes".MotionToPLC.Stauts.DancerMain.Error;
END_REGION

REGION Network 77: Commands ReelCutMain
   RUNG wire#powerrail
      Contact( #TRUE )
      wire#w1
      Contact( "Unit1.Em3.ControlNodes".webGuid."step".action[231] )
      Coil( "Unit1.MotionNodes".PLCToMotion.Commands.ReelCutMain.Calculate )
   END_RUNG
   RUNG wire#w1
      Contact( "Unit1.Em3.ControlNodes".webGuid."step".action[331] )
      Coil( "Unit1.MotionNodes".PLCToMotion.Commands.ReelCutMain.OneCell )
   END_RUNG
   RUNG wire#w1
      Contact( "Unit1.Em3.ControlNodes".webGuid."step".action[431] )
      Coil( "Unit1.MotionNodes".PLCToMotion.Commands.ReelCutMain.FullStep )
   END_RUNG
   RUNG wire#w1
      Contact( "Unit1.Em3.ControlNodes".webGuid."step".action[531] )
      Coil( "Unit1.MotionNodes".PLCToMotion.Commands.ReelCutMain.Auto )
   END_RUNG
   RUNG wire#w1
      Contact( "Unit1.Em3.ControlNodes".webGuid."step".action[631] )
      Coil( "Unit1.MotionNodes".PLCToMotion.Commands.ReelCutMain.SemiStep )
   END_RUNG
   RUNG wire#w1
      I_Contact( "Unit1.Em3.ControlNodes".webGuid."step".action[211] )
      I_Contact( "Unit1.Em3.ControlNodes".webGuid."step".action[311] )
      I_Contact( "Unit1.Em3.ControlNodes".webGuid."step".action[411] )
      I_Contact( "Unit1.Em3.ControlNodes".webGuid."step".action[511] )
      I_Contact( "Unit1.Em3.ControlNodes".webGuid."step".action[611] )
      I_Contact( "Unit1.Em3.ControlNodes".webGuid."step".action[711] )
      Not()
      Coil( "Unit1.MotionNodes".PLCToMotion.Commands.ReelCutMain.CycleStop )
   END_RUNG
   RUNG wire#w1
      Contact( "Unit1.Em3.ControlNodes".webGuid."step".action[811] )
      Coil( "Unit1.MotionNodes".PLCToMotion.Commands.ReelCutMain.FastStop )
   END_RUNG
   RUNG wire#w1
      Contact( #statUnitStatus.acknowledgeActive )
      wire#w2
      Contact( "Unit1.MotionNodes".MotionToPLC.Stauts.ReelCutMain.Error )
      Coil( "Unit1.MotionNodes".PLCToMotion.Commands.ReelCutMain.Reset )
   END_RUNG
   RUNG wire#w1
      Contact( #statUnitStatus.state.resetting )
   END_RUNG wire#w2
   // the same network as SCL:
   "Unit1.MotionNodes".PLCToMotion.Commands.ReelCutMain.Calculate := #TRUE AND "Unit1.Em3.ControlNodes".webGuid."step".action[231];
   "Unit1.MotionNodes".PLCToMotion.Commands.ReelCutMain.OneCell := #TRUE AND "Unit1.Em3.ControlNodes".webGuid."step".action[331];
   "Unit1.MotionNodes".PLCToMotion.Commands.ReelCutMain.FullStep := #TRUE AND "Unit1.Em3.ControlNodes".webGuid."step".action[431];
   "Unit1.MotionNodes".PLCToMotion.Commands.ReelCutMain.Auto := #TRUE AND "Unit1.Em3.ControlNodes".webGuid."step".action[531];
   "Unit1.MotionNodes".PLCToMotion.Commands.ReelCutMain.SemiStep := #TRUE AND "Unit1.Em3.ControlNodes".webGuid."step".action[631];
   "Unit1.MotionNodes".PLCToMotion.Commands.ReelCutMain.CycleStop := NOT (#TRUE AND NOT "Unit1.Em3.ControlNodes".webGuid."step".action[211] AND NOT "Unit1.Em3.ControlNodes".webGuid."step".action[311] AND NOT "Unit1.Em3.ControlNodes".webGuid."step".action[411] AND NOT "Unit1.Em3.ControlNodes".webGuid."step".action[511] AND NOT "Unit1.Em3.ControlNodes".webGuid."step".action[611] AND NOT "Unit1.Em3.ControlNodes".webGuid."step".action[711]);
   "Unit1.MotionNodes".PLCToMotion.Commands.ReelCutMain.FastStop := #TRUE AND "Unit1.Em3.ControlNodes".webGuid."step".action[811];
   "Unit1.MotionNodes".PLCToMotion.Commands.ReelCutMain.Reset := #TRUE AND (#statUnitStatus.acknowledgeActive OR #statUnitStatus.state.resetting) AND "Unit1.MotionNodes".MotionToPLC.Stauts.ReelCutMain.Error;
END_REGION

REGION Network 78: Commands MeasureIMain
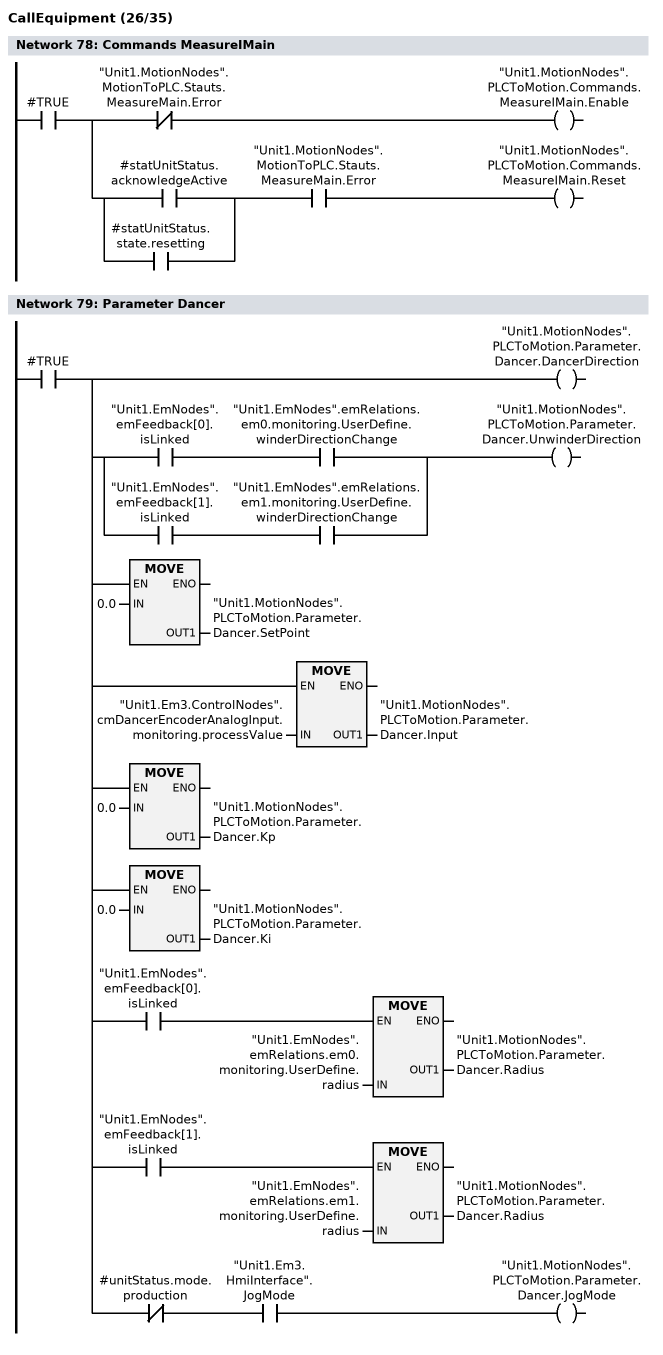
   RUNG wire#powerrail
      Contact( #TRUE )
      wire#w1
      I_Contact( "Unit1.MotionNodes".MotionToPLC.Stauts.MeasureMain.Error )
      Coil( "Unit1.MotionNodes".PLCToMotion.Commands.MeasureIMain.Enable )
   END_RUNG
   RUNG wire#w1
      Contact( #statUnitStatus.acknowledgeActive )
      wire#w2
      Contact( "Unit1.MotionNodes".MotionToPLC.Stauts.MeasureMain.Error )
      Coil( "Unit1.MotionNodes".PLCToMotion.Commands.MeasureIMain.Reset )
   END_RUNG
   RUNG wire#w1
      Contact( #statUnitStatus.state.resetting )
   END_RUNG wire#w2
   // the same network as SCL:
   "Unit1.MotionNodes".PLCToMotion.Commands.MeasureIMain.Enable := #TRUE AND NOT "Unit1.MotionNodes".MotionToPLC.Stauts.MeasureMain.Error;
   "Unit1.MotionNodes".PLCToMotion.Commands.MeasureIMain.Reset := #TRUE AND (#statUnitStatus.acknowledgeActive OR #statUnitStatus.state.resetting) AND "Unit1.MotionNodes".MotionToPLC.Stauts.MeasureMain.Error;
END_REGION

REGION Network 79: Parameter Dancer
   RUNG wire#powerrail
      Contact( #TRUE )
      wire#w1
      Coil( "Unit1.MotionNodes".PLCToMotion.Parameter.Dancer.DancerDirection )
   END_RUNG
   RUNG wire#w1
      Contact( "Unit1.EmNodes".emFeedback[0].isLinked )
      Contact( "Unit1.EmNodes".emRelations.em0.monitoring.UserDefine.winderDirectionChange )
      wire#w2
      Coil( "Unit1.MotionNodes".PLCToMotion.Parameter.Dancer.UnwinderDirection )
   END_RUNG
   RUNG wire#w1
      Contact( "Unit1.EmNodes".emFeedback[1].isLinked )
      Contact( "Unit1.EmNodes".emRelations.em1.monitoring.UserDefine.winderDirectionChange )
   END_RUNG wire#w2
   RUNG wire#w1
      Move(in := 0.0, out1 => "Unit1.MotionNodes".PLCToMotion.Parameter.Dancer.SetPoint)
   END_RUNG
   RUNG wire#w1
      Move(in := "Unit1.Em3.ControlNodes".cmDancerEncoderAnalogInput.monitoring.processValue, out1 => "Unit1.MotionNodes".PLCToMotion.Parameter.Dancer.Input)
   END_RUNG
   RUNG wire#w1
      Move(in := 0.0, out1 => "Unit1.MotionNodes".PLCToMotion.Parameter.Dancer.Kp)
   END_RUNG
   RUNG wire#w1
      Move(in := 0.0, out1 => "Unit1.MotionNodes".PLCToMotion.Parameter.Dancer.Ki)
   END_RUNG
   RUNG wire#w1
      Contact( "Unit1.EmNodes".emFeedback[0].isLinked )
      Move(in := "Unit1.EmNodes".emRelations.em0.monitoring.UserDefine.radius, out1 => "Unit1.MotionNodes".PLCToMotion.Parameter.Dancer.Radius)
   END_RUNG
   RUNG wire#w1
      Contact( "Unit1.EmNodes".emFeedback[1].isLinked )
      Move(in := "Unit1.EmNodes".emRelations.em1.monitoring.UserDefine.radius, out1 => "Unit1.MotionNodes".PLCToMotion.Parameter.Dancer.Radius)
   END_RUNG
   RUNG wire#w1
      I_Contact( #unitStatus.mode.production )
      Contact( "Unit1.Em3.HmiInterface".JogMode )
      Coil( "Unit1.MotionNodes".PLCToMotion.Parameter.Dancer.JogMode )
   END_RUNG
   // the same network as SCL:
   "Unit1.MotionNodes".PLCToMotion.Parameter.Dancer.DancerDirection := #TRUE;
   "Unit1.MotionNodes".PLCToMotion.Parameter.Dancer.UnwinderDirection := #TRUE AND (("Unit1.EmNodes".emFeedback[0].isLinked AND "Unit1.EmNodes".emRelations.em0.monitoring.UserDefine.winderDirectionChange) OR ("Unit1.EmNodes".emFeedback[1].isLinked AND "Unit1.EmNodes".emRelations.em1.monitoring.UserDefine.winderDirectionChange));
   IF #TRUE THEN
       "Unit1.MotionNodes".PLCToMotion.Parameter.Dancer.SetPoint := 0.0;
       "Unit1.MotionNodes".PLCToMotion.Parameter.Dancer.Input := "Unit1.Em3.ControlNodes".cmDancerEncoderAnalogInput.monitoring.processValue;
       "Unit1.MotionNodes".PLCToMotion.Parameter.Dancer.Kp := 0.0;
       "Unit1.MotionNodes".PLCToMotion.Parameter.Dancer.Ki := 0.0;
   END_IF;
   IF #TRUE AND "Unit1.EmNodes".emFeedback[0].isLinked THEN
       "Unit1.MotionNodes".PLCToMotion.Parameter.Dancer.Radius := "Unit1.EmNodes".emRelations.em0.monitoring.UserDefine.radius;
   END_IF;
   IF #TRUE AND "Unit1.EmNodes".emFeedback[1].isLinked THEN
       "Unit1.MotionNodes".PLCToMotion.Parameter.Dancer.Radius := "Unit1.EmNodes".emRelations.em1.monitoring.UserDefine.radius;
   END_IF;
   "Unit1.MotionNodes".PLCToMotion.Parameter.Dancer.JogMode := #TRUE AND NOT #unitStatus.mode.production AND "Unit1.Em3.HmiInterface".JogMode;
END_REGION

REGION Network 80: Parameter ReelCutMain Global
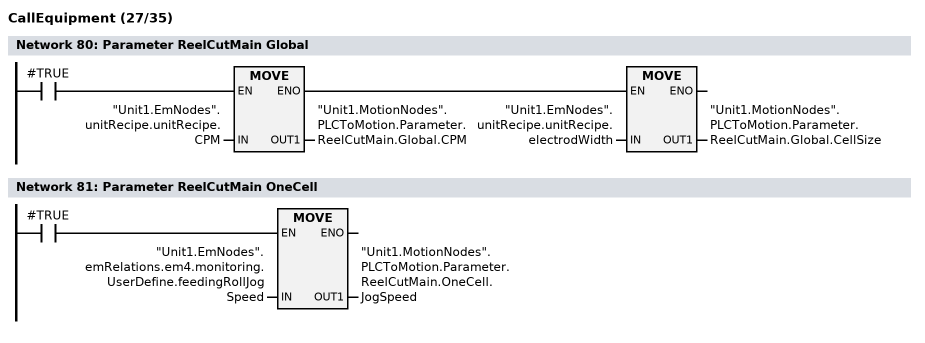
   RUNG wire#powerrail
      Contact( #TRUE )
      Move(in := "Unit1.EmNodes".unitRecipe.unitRecipe.CPM, out1 => "Unit1.MotionNodes".PLCToMotion.Parameter.ReelCutMain.Global.CPM)
      Move(in := "Unit1.EmNodes".unitRecipe.unitRecipe.electrodWidth, out1 => "Unit1.MotionNodes".PLCToMotion.Parameter.ReelCutMain.Global.CellSize)
   END_RUNG
   // the same network as SCL:
   IF #TRUE THEN
       "Unit1.MotionNodes".PLCToMotion.Parameter.ReelCutMain.Global.CPM := "Unit1.EmNodes".unitRecipe.unitRecipe.CPM;
       "Unit1.MotionNodes".PLCToMotion.Parameter.ReelCutMain.Global.CellSize := "Unit1.EmNodes".unitRecipe.unitRecipe.electrodWidth;
   END_IF;
END_REGION

REGION Network 81: Parameter ReelCutMain OneCell
   RUNG wire#powerrail
      Contact( #TRUE )
      Move(in := "Unit1.EmNodes".emRelations.em4.monitoring.UserDefine.feedingRollJogSpeed, out1 => "Unit1.MotionNodes".PLCToMotion.Parameter.ReelCutMain.OneCell.JogSpeed)
   END_RUNG
   // the same network as SCL:
   IF #TRUE THEN
       "Unit1.MotionNodes".PLCToMotion.Parameter.ReelCutMain.OneCell.JogSpeed := "Unit1.EmNodes".emRelations.em4.monitoring.UserDefine.feedingRollJogSpeed;
   END_IF;
END_REGION

REGION Network 82: Parameter ReelCutMain StepAuto
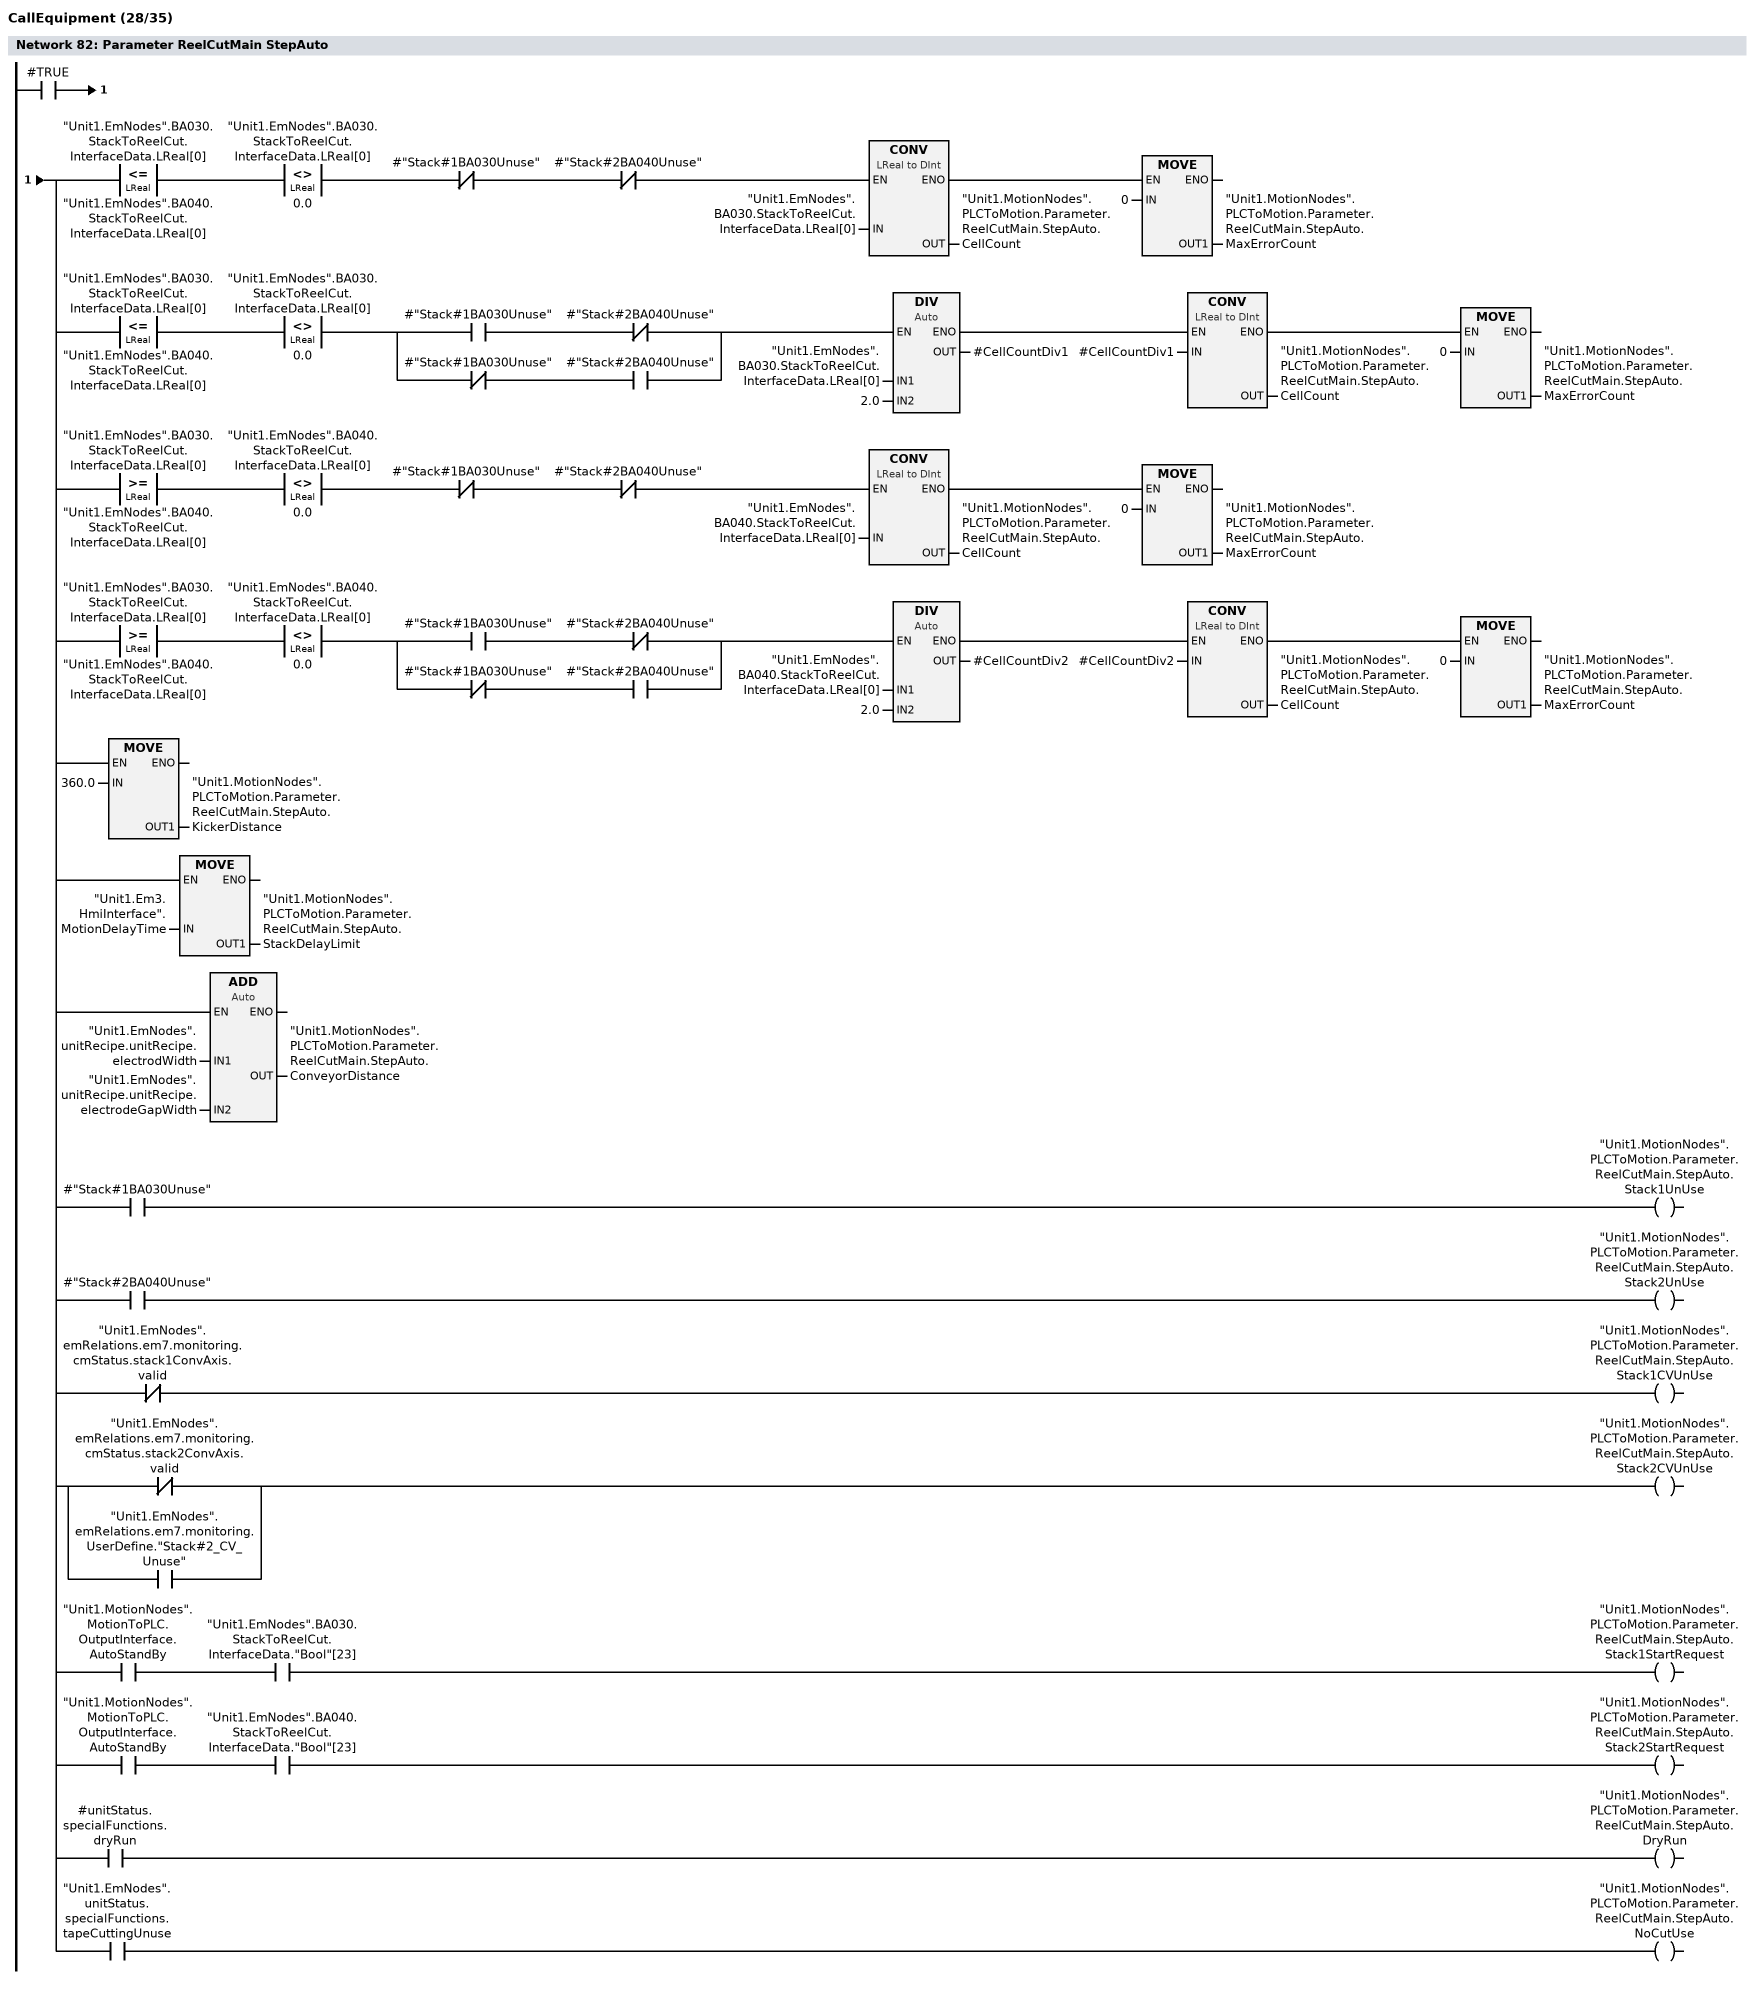
   RUNG wire#powerrail
      Contact( #TRUE )
      wire#w1
      { S7_Templates := "SrcType := LReal" } LE_Contact(in1 := "Unit1.EmNodes".BA030.StackToReelCut.InterfaceData.LReal[0], in2 := "Unit1.EmNodes".BA040.StackToReelCut.InterfaceData.LReal[0])
      { S7_Templates := "SrcType := LReal" } NE_Contact(in1 := "Unit1.EmNodes".BA030.StackToReelCut.InterfaceData.LReal[0], in2 := 0.0)
      I_Contact( #"Stack#1BA030Unuse" )
      I_Contact( #"Stack#2BA040Unuse" )
      { S7_Templates := "[SrcType := LReal, DestType := DInt]" } Convert(in := "Unit1.EmNodes".BA030.StackToReelCut.InterfaceData.LReal[0], out => "Unit1.MotionNodes".PLCToMotion.Parameter.ReelCutMain.StepAuto.CellCount)
      Move(in := 0, out1 => "Unit1.MotionNodes".PLCToMotion.Parameter.ReelCutMain.StepAuto.MaxErrorCount)
   END_RUNG
   RUNG wire#w1
      { S7_Templates := "SrcType := LReal" } LE_Contact(in1 := "Unit1.EmNodes".BA030.StackToReelCut.InterfaceData.LReal[0], in2 := "Unit1.EmNodes".BA040.StackToReelCut.InterfaceData.LReal[0])
      { S7_Templates := "SrcType := LReal" } NE_Contact(in1 := "Unit1.EmNodes".BA030.StackToReelCut.InterfaceData.LReal[0], in2 := 0.0)
      wire#w2
      Contact( #"Stack#1BA030Unuse" )
      I_Contact( #"Stack#2BA040Unuse" )
      wire#w3
      Div(in1 := "Unit1.EmNodes".BA030.StackToReelCut.InterfaceData.LReal[0], in2 := 2.0, out => #CellCountDiv1)
      { S7_Templates := "[SrcType := LReal, DestType := DInt]" } Convert(in := #CellCountDiv1, out => "Unit1.MotionNodes".PLCToMotion.Parameter.ReelCutMain.StepAuto.CellCount)
      Move(in := 0, out1 => "Unit1.MotionNodes".PLCToMotion.Parameter.ReelCutMain.StepAuto.MaxErrorCount)
   END_RUNG
   RUNG wire#w2
      I_Contact( #"Stack#1BA030Unuse" )
      Contact( #"Stack#2BA040Unuse" )
   END_RUNG wire#w3
   RUNG wire#w1
      { S7_Templates := "SrcType := LReal" } GE_Contact(in1 := "Unit1.EmNodes".BA030.StackToReelCut.InterfaceData.LReal[0], in2 := "Unit1.EmNodes".BA040.StackToReelCut.InterfaceData.LReal[0])
      { S7_Templates := "SrcType := LReal" } NE_Contact(in1 := "Unit1.EmNodes".BA040.StackToReelCut.InterfaceData.LReal[0], in2 := 0.0)
      I_Contact( #"Stack#1BA030Unuse" )
      I_Contact( #"Stack#2BA040Unuse" )
      { S7_Templates := "[SrcType := LReal, DestType := DInt]" } Convert(in := "Unit1.EmNodes".BA040.StackToReelCut.InterfaceData.LReal[0], out => "Unit1.MotionNodes".PLCToMotion.Parameter.ReelCutMain.StepAuto.CellCount)
      Move(in := 0, out1 => "Unit1.MotionNodes".PLCToMotion.Parameter.ReelCutMain.StepAuto.MaxErrorCount)
   END_RUNG
   RUNG wire#w1
      { S7_Templates := "SrcType := LReal" } GE_Contact(in1 := "Unit1.EmNodes".BA030.StackToReelCut.InterfaceData.LReal[0], in2 := "Unit1.EmNodes".BA040.StackToReelCut.InterfaceData.LReal[0])
      { S7_Templates := "SrcType := LReal" } NE_Contact(in1 := "Unit1.EmNodes".BA040.StackToReelCut.InterfaceData.LReal[0], in2 := 0.0)
      wire#w4
      Contact( #"Stack#1BA030Unuse" )
      I_Contact( #"Stack#2BA040Unuse" )
      wire#w5
      Div(in1 := "Unit1.EmNodes".BA040.StackToReelCut.InterfaceData.LReal[0], in2 := 2.0, out => #CellCountDiv2)
      { S7_Templates := "[SrcType := LReal, DestType := DInt]" } Convert(in := #CellCountDiv2, out => "Unit1.MotionNodes".PLCToMotion.Parameter.ReelCutMain.StepAuto.CellCount)
      Move(in := 0, out1 => "Unit1.MotionNodes".PLCToMotion.Parameter.ReelCutMain.StepAuto.MaxErrorCount)
   END_RUNG
   RUNG wire#w4
      I_Contact( #"Stack#1BA030Unuse" )
      Contact( #"Stack#2BA040Unuse" )
   END_RUNG wire#w5
   RUNG wire#w1
      Move(in := 360.0, out1 => "Unit1.MotionNodes".PLCToMotion.Parameter.ReelCutMain.StepAuto.KickerDistance)
   END_RUNG
   RUNG wire#w1
      Move(in := "Unit1.Em3.HmiInterface".MotionDelayTime, out1 => "Unit1.MotionNodes".PLCToMotion.Parameter.ReelCutMain.StepAuto.StackDelayLimit)
   END_RUNG
   RUNG wire#w1
      Add(in1 := "Unit1.EmNodes".unitRecipe.unitRecipe.electrodWidth, in2 := "Unit1.EmNodes".unitRecipe.unitRecipe.electrodeGapWidth, out => "Unit1.MotionNodes".PLCToMotion.Parameter.ReelCutMain.StepAuto.ConveyorDistance)
   END_RUNG
   RUNG wire#w1
      Contact( #"Stack#1BA030Unuse" )
      Coil( "Unit1.MotionNodes".PLCToMotion.Parameter.ReelCutMain.StepAuto.Stack1UnUse )
   END_RUNG
   RUNG wire#w1
      Contact( #"Stack#2BA040Unuse" )
      Coil( "Unit1.MotionNodes".PLCToMotion.Parameter.ReelCutMain.StepAuto.Stack2UnUse )
   END_RUNG
   RUNG wire#w1
      I_Contact( "Unit1.EmNodes".emRelations.em7.monitoring.cmStatus.stack1ConvAxis.valid )
      Coil( "Unit1.MotionNodes".PLCToMotion.Parameter.ReelCutMain.StepAuto.Stack1CVUnUse )
   END_RUNG
   RUNG wire#w1
      I_Contact( "Unit1.EmNodes".emRelations.em7.monitoring.cmStatus.stack2ConvAxis.valid )
      wire#w6
      Coil( "Unit1.MotionNodes".PLCToMotion.Parameter.ReelCutMain.StepAuto.Stack2CVUnUse )
   END_RUNG
   RUNG wire#w1
      Contact( "Unit1.EmNodes".emRelations.em7.monitoring.UserDefine."Stack#2_CV_Unuse" )
   END_RUNG wire#w6
   RUNG wire#w1
      Contact( "Unit1.MotionNodes".MotionToPLC.OutputInterface.AutoStandBy )
      Contact( "Unit1.EmNodes".BA030.StackToReelCut.InterfaceData."Bool"[23] )
      Coil( "Unit1.MotionNodes".PLCToMotion.Parameter.ReelCutMain.StepAuto.Stack1StartRequest )
   END_RUNG
   RUNG wire#w1
      Contact( "Unit1.MotionNodes".MotionToPLC.OutputInterface.AutoStandBy )
      Contact( "Unit1.EmNodes".BA040.StackToReelCut.InterfaceData."Bool"[23] )
      Coil( "Unit1.MotionNodes".PLCToMotion.Parameter.ReelCutMain.StepAuto.Stack2StartRequest )
   END_RUNG
   RUNG wire#w1
      Contact( #unitStatus.specialFunctions.dryRun )
      Coil( "Unit1.MotionNodes".PLCToMotion.Parameter.ReelCutMain.StepAuto.DryRun )
   END_RUNG
   RUNG wire#w1
      Contact( "Unit1.EmNodes".unitStatus.specialFunctions.tapeCuttingUnuse )
      Coil( "Unit1.MotionNodes".PLCToMotion.Parameter.ReelCutMain.StepAuto.NoCutUse )
   END_RUNG
   // the same network as SCL:
   IF #TRUE AND ("Unit1.EmNodes".BA030.StackToReelCut.InterfaceData.LReal[0] <= "Unit1.EmNodes".BA040.StackToReelCut.InterfaceData.LReal[0]) AND ("Unit1.EmNodes".BA030.StackToReelCut.InterfaceData.LReal[0] <> 0.0) AND NOT #"Stack#1BA030Unuse" AND NOT #"Stack#2BA040Unuse" THEN
       "Unit1.MotionNodes".PLCToMotion.Parameter.ReelCutMain.StepAuto.CellCount := LREAL_TO_DINT("Unit1.EmNodes".BA030.StackToReelCut.InterfaceData.LReal[0]);
       "Unit1.MotionNodes".PLCToMotion.Parameter.ReelCutMain.StepAuto.MaxErrorCount := 0;
   END_IF;
   IF #TRUE AND ("Unit1.EmNodes".BA030.StackToReelCut.InterfaceData.LReal[0] <= "Unit1.EmNodes".BA040.StackToReelCut.InterfaceData.LReal[0]) AND ("Unit1.EmNodes".BA030.StackToReelCut.InterfaceData.LReal[0] <> 0.0) AND ((#"Stack#1BA030Unuse" AND NOT #"Stack#2BA040Unuse") OR (NOT #"Stack#1BA030Unuse" AND #"Stack#2BA040Unuse")) THEN
       #CellCountDiv1 := "Unit1.EmNodes".BA030.StackToReelCut.InterfaceData.LReal[0] / 2.0;
       "Unit1.MotionNodes".PLCToMotion.Parameter.ReelCutMain.StepAuto.CellCount := LREAL_TO_DINT(#CellCountDiv1);
       "Unit1.MotionNodes".PLCToMotion.Parameter.ReelCutMain.StepAuto.MaxErrorCount := 0;
   END_IF;
   IF #TRUE AND ("Unit1.EmNodes".BA030.StackToReelCut.InterfaceData.LReal[0] >= "Unit1.EmNodes".BA040.StackToReelCut.InterfaceData.LReal[0]) AND ("Unit1.EmNodes".BA040.StackToReelCut.InterfaceData.LReal[0] <> 0.0) AND NOT #"Stack#1BA030Unuse" AND NOT #"Stack#2BA040Unuse" THEN
       "Unit1.MotionNodes".PLCToMotion.Parameter.ReelCutMain.StepAuto.CellCount := LREAL_TO_DINT("Unit1.EmNodes".BA040.StackToReelCut.InterfaceData.LReal[0]);
       "Unit1.MotionNodes".PLCToMotion.Parameter.ReelCutMain.StepAuto.MaxErrorCount := 0;
   END_IF;
   IF #TRUE AND ("Unit1.EmNodes".BA030.StackToReelCut.InterfaceData.LReal[0] >= "Unit1.EmNodes".BA040.StackToReelCut.InterfaceData.LReal[0]) AND ("Unit1.EmNodes".BA040.StackToReelCut.InterfaceData.LReal[0] <> 0.0) AND ((#"Stack#1BA030Unuse" AND NOT #"Stack#2BA040Unuse") OR (NOT #"Stack#1BA030Unuse" AND #"Stack#2BA040Unuse")) THEN
       #CellCountDiv2 := "Unit1.EmNodes".BA040.StackToReelCut.InterfaceData.LReal[0] / 2.0;
       "Unit1.MotionNodes".PLCToMotion.Parameter.ReelCutMain.StepAuto.CellCount := LREAL_TO_DINT(#CellCountDiv2);
       "Unit1.MotionNodes".PLCToMotion.Parameter.ReelCutMain.StepAuto.MaxErrorCount := 0;
   END_IF;
   IF #TRUE THEN
       "Unit1.MotionNodes".PLCToMotion.Parameter.ReelCutMain.StepAuto.KickerDistance := 360.0;
       "Unit1.MotionNodes".PLCToMotion.Parameter.ReelCutMain.StepAuto.StackDelayLimit := "Unit1.Em3.HmiInterface".MotionDelayTime;
       "Unit1.MotionNodes".PLCToMotion.Parameter.ReelCutMain.StepAuto.ConveyorDistance := "Unit1.EmNodes".unitRecipe.unitRecipe.electrodWidth + "Unit1.EmNodes".unitRecipe.unitRecipe.electrodeGapWidth;
   END_IF;
   "Unit1.MotionNodes".PLCToMotion.Parameter.ReelCutMain.StepAuto.Stack1UnUse := #TRUE AND #"Stack#1BA030Unuse";
   "Unit1.MotionNodes".PLCToMotion.Parameter.ReelCutMain.StepAuto.Stack2UnUse := #TRUE AND #"Stack#2BA040Unuse";
   "Unit1.MotionNodes".PLCToMotion.Parameter.ReelCutMain.StepAuto.Stack1CVUnUse := #TRUE AND NOT "Unit1.EmNodes".emRelations.em7.monitoring.cmStatus.stack1ConvAxis.valid;
   "Unit1.MotionNodes".PLCToMotion.Parameter.ReelCutMain.StepAuto.Stack2CVUnUse := #TRUE AND (NOT "Unit1.EmNodes".emRelations.em7.monitoring.cmStatus.stack2ConvAxis.valid OR "Unit1.EmNodes".emRelations.em7.monitoring.UserDefine."Stack#2_CV_Unuse");
   "Unit1.MotionNodes".PLCToMotion.Parameter.ReelCutMain.StepAuto.Stack1StartRequest := #TRUE AND "Unit1.MotionNodes".MotionToPLC.OutputInterface.AutoStandBy AND "Unit1.EmNodes".BA030.StackToReelCut.InterfaceData."Bool"[23];
   "Unit1.MotionNodes".PLCToMotion.Parameter.ReelCutMain.StepAuto.Stack2StartRequest := #TRUE AND "Unit1.MotionNodes".MotionToPLC.OutputInterface.AutoStandBy AND "Unit1.EmNodes".BA040.StackToReelCut.InterfaceData."Bool"[23];
   "Unit1.MotionNodes".PLCToMotion.Parameter.ReelCutMain.StepAuto.DryRun := #TRUE AND #unitStatus.specialFunctions.dryRun;
   "Unit1.MotionNodes".PLCToMotion.Parameter.ReelCutMain.StepAuto.NoCutUse := #TRUE AND "Unit1.EmNodes".unitStatus.specialFunctions.tapeCuttingUnuse;
END_REGION

REGION Network 83: Parameter ReelCutMain Calculate
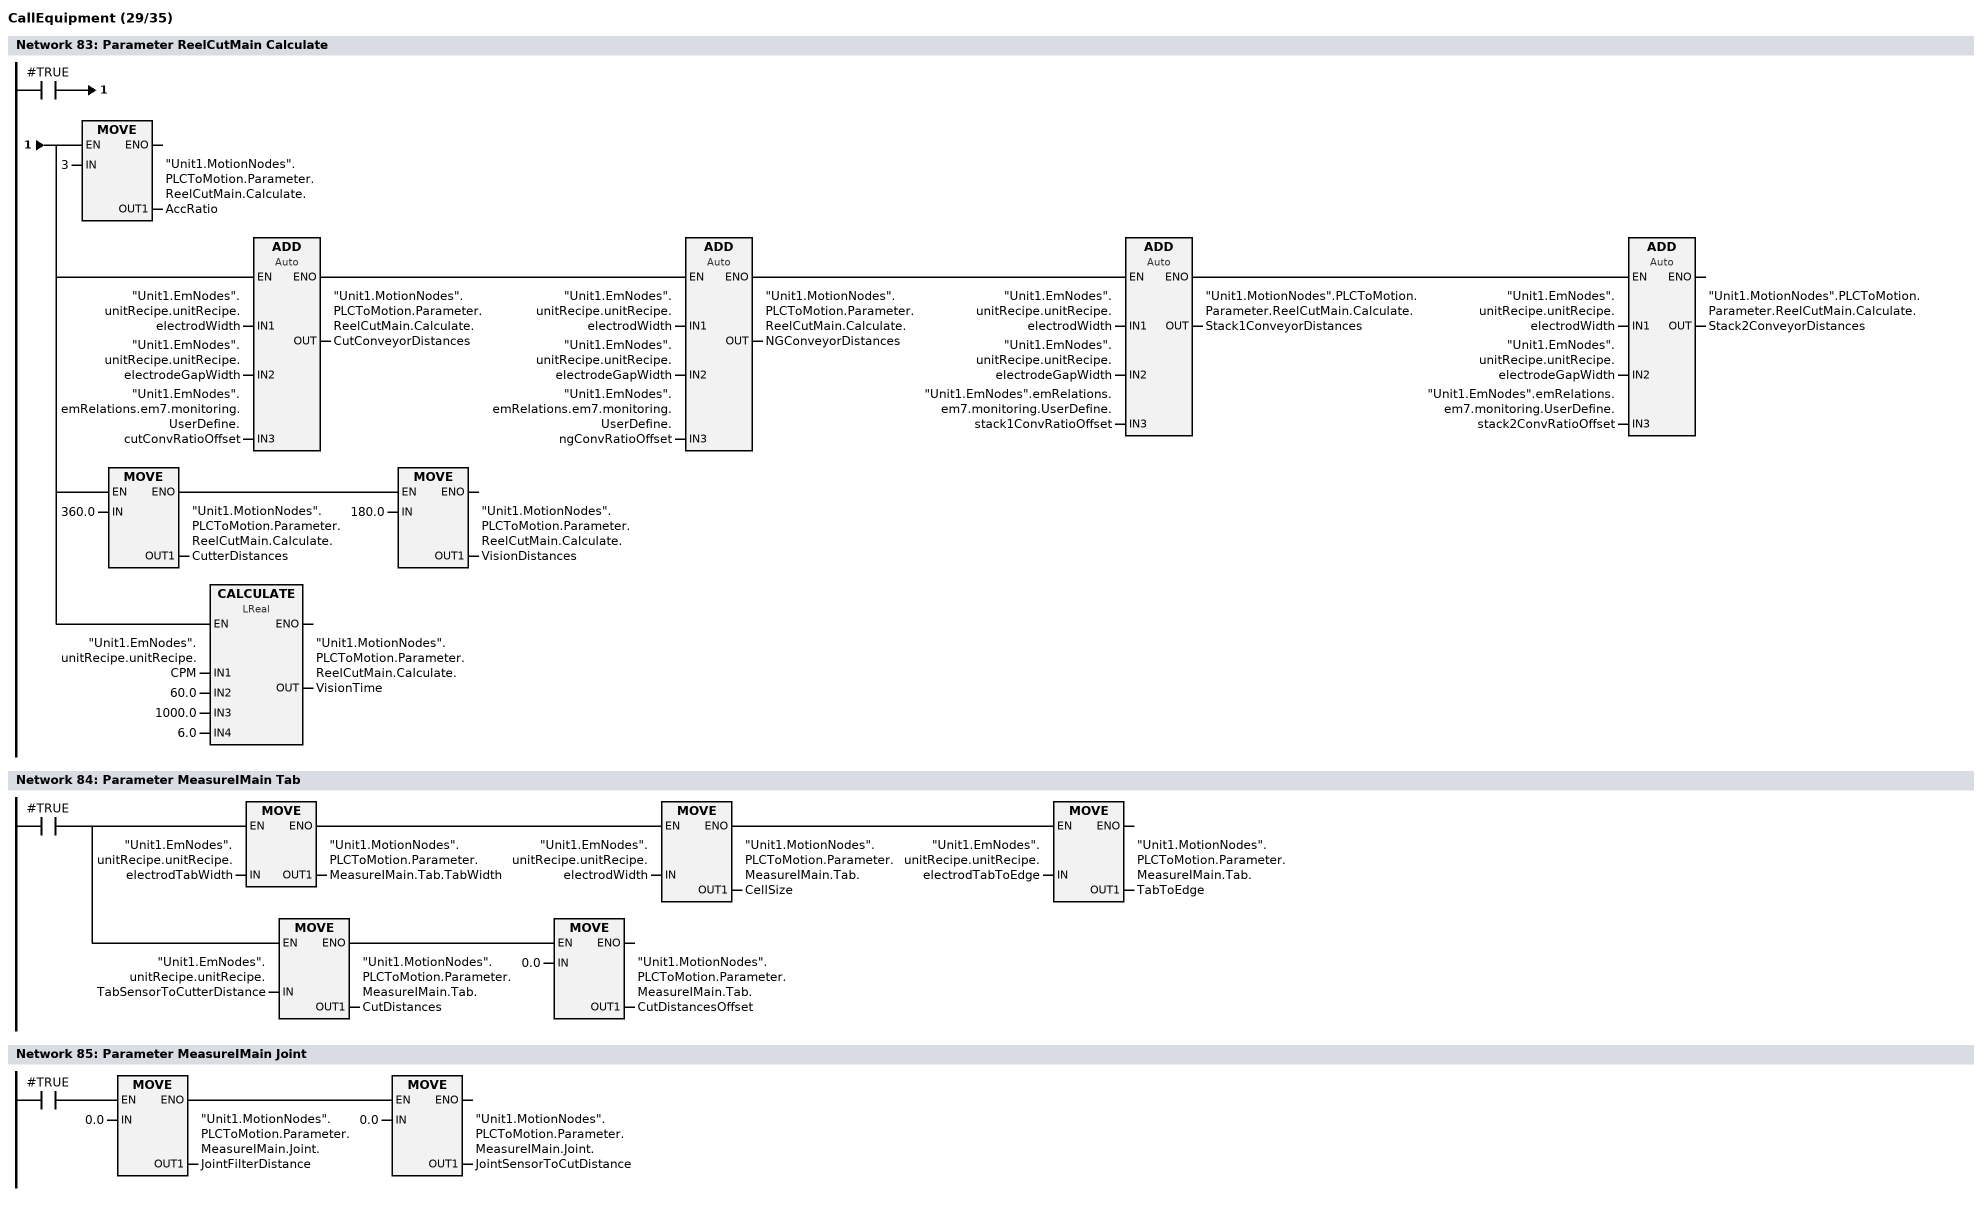
   RUNG wire#powerrail
      Contact( #TRUE )
      wire#w1
      Move(in := 3, out1 => "Unit1.MotionNodes".PLCToMotion.Parameter.ReelCutMain.Calculate.AccRatio)
   END_RUNG
   RUNG wire#w1
      Add(in1 := "Unit1.EmNodes".unitRecipe.unitRecipe.electrodWidth, in2 := "Unit1.EmNodes".unitRecipe.unitRecipe.electrodeGapWidth, in3 := "Unit1.EmNodes".emRelations.em7.monitoring.UserDefine.cutConvRatioOffset, out => "Unit1.MotionNodes".PLCToMotion.Parameter.ReelCutMain.Calculate.CutConveyorDistances)
      Add(in1 := "Unit1.EmNodes".unitRecipe.unitRecipe.electrodWidth, in2 := "Unit1.EmNodes".unitRecipe.unitRecipe.electrodeGapWidth, in3 := "Unit1.EmNodes".emRelations.em7.monitoring.UserDefine.ngConvRatioOffset, out => "Unit1.MotionNodes".PLCToMotion.Parameter.ReelCutMain.Calculate.NGConveyorDistances)
      Add(in1 := "Unit1.EmNodes".unitRecipe.unitRecipe.electrodWidth, in2 := "Unit1.EmNodes".unitRecipe.unitRecipe.electrodeGapWidth, in3 := "Unit1.EmNodes".emRelations.em7.monitoring.UserDefine.stack1ConvRatioOffset, out => "Unit1.MotionNodes".PLCToMotion.Parameter.ReelCutMain.Calculate.Stack1ConveyorDistances)
      Add(in1 := "Unit1.EmNodes".unitRecipe.unitRecipe.electrodWidth, in2 := "Unit1.EmNodes".unitRecipe.unitRecipe.electrodeGapWidth, in3 := "Unit1.EmNodes".emRelations.em7.monitoring.UserDefine.stack2ConvRatioOffset, out => "Unit1.MotionNodes".PLCToMotion.Parameter.ReelCutMain.Calculate.Stack2ConveyorDistances)
   END_RUNG
   RUNG wire#w1
      Move(in := 360.0, out1 => "Unit1.MotionNodes".PLCToMotion.Parameter.ReelCutMain.Calculate.CutterDistances)
      Move(in := 180.0, out1 => "Unit1.MotionNodes".PLCToMotion.Parameter.ReelCutMain.Calculate.VisionDistances)
   END_RUNG
   RUNG wire#w1
      { S7_Templates := "SrcType := LReal"; S7_Expression := "(IN2/IN1)*IN3/IN4" } Calculate(in1 := "Unit1.EmNodes".unitRecipe.unitRecipe.CPM, in2 := 60.0, in3 := 1000.0, in4 := 6.0, out => "Unit1.MotionNodes".PLCToMotion.Parameter.ReelCutMain.Calculate.VisionTime)
   END_RUNG
   // the same network as SCL:
   IF #TRUE THEN
       "Unit1.MotionNodes".PLCToMotion.Parameter.ReelCutMain.Calculate.AccRatio := 3;
       "Unit1.MotionNodes".PLCToMotion.Parameter.ReelCutMain.Calculate.CutConveyorDistances := "Unit1.EmNodes".unitRecipe.unitRecipe.electrodWidth + "Unit1.EmNodes".unitRecipe.unitRecipe.electrodeGapWidth + "Unit1.EmNodes".emRelations.em7.monitoring.UserDefine.cutConvRatioOffset;
       "Unit1.MotionNodes".PLCToMotion.Parameter.ReelCutMain.Calculate.NGConveyorDistances := "Unit1.EmNodes".unitRecipe.unitRecipe.electrodWidth + "Unit1.EmNodes".unitRecipe.unitRecipe.electrodeGapWidth + "Unit1.EmNodes".emRelations.em7.monitoring.UserDefine.ngConvRatioOffset;
       "Unit1.MotionNodes".PLCToMotion.Parameter.ReelCutMain.Calculate.Stack1ConveyorDistances := "Unit1.EmNodes".unitRecipe.unitRecipe.electrodWidth + "Unit1.EmNodes".unitRecipe.unitRecipe.electrodeGapWidth + "Unit1.EmNodes".emRelations.em7.monitoring.UserDefine.stack1ConvRatioOffset;
       "Unit1.MotionNodes".PLCToMotion.Parameter.ReelCutMain.Calculate.Stack2ConveyorDistances := "Unit1.EmNodes".unitRecipe.unitRecipe.electrodWidth + "Unit1.EmNodes".unitRecipe.unitRecipe.electrodeGapWidth + "Unit1.EmNodes".emRelations.em7.monitoring.UserDefine.stack2ConvRatioOffset;
       "Unit1.MotionNodes".PLCToMotion.Parameter.ReelCutMain.Calculate.CutterDistances := 360.0;
       "Unit1.MotionNodes".PLCToMotion.Parameter.ReelCutMain.Calculate.VisionDistances := 180.0;
       "Unit1.MotionNodes".PLCToMotion.Parameter.ReelCutMain.Calculate.VisionTime := (60.0/"Unit1.EmNodes".unitRecipe.unitRecipe.CPM)*1000.0/6.0;
   END_IF;
END_REGION

REGION Network 84: Parameter MeasureIMain Tab
   RUNG wire#powerrail
      Contact( #TRUE )
      wire#w1
      Move(in := "Unit1.EmNodes".unitRecipe.unitRecipe.electrodTabWidth, out1 => "Unit1.MotionNodes".PLCToMotion.Parameter.MeasureIMain.Tab.TabWidth)
      Move(in := "Unit1.EmNodes".unitRecipe.unitRecipe.electrodWidth, out1 => "Unit1.MotionNodes".PLCToMotion.Parameter.MeasureIMain.Tab.CellSize)
      Move(in := "Unit1.EmNodes".unitRecipe.unitRecipe.electrodTabToEdge, out1 => "Unit1.MotionNodes".PLCToMotion.Parameter.MeasureIMain.Tab.TabToEdge)
   END_RUNG
   RUNG wire#w1
      Move(in := "Unit1.EmNodes".unitRecipe.unitRecipe.TabSensorToCutterDistance, out1 => "Unit1.MotionNodes".PLCToMotion.Parameter.MeasureIMain.Tab.CutDistances)
      Move(in := 0.0, out1 => "Unit1.MotionNodes".PLCToMotion.Parameter.MeasureIMain.Tab.CutDistancesOffset)
   END_RUNG
   // the same network as SCL:
   IF #TRUE THEN
       "Unit1.MotionNodes".PLCToMotion.Parameter.MeasureIMain.Tab.TabWidth := "Unit1.EmNodes".unitRecipe.unitRecipe.electrodTabWidth;
       "Unit1.MotionNodes".PLCToMotion.Parameter.MeasureIMain.Tab.CellSize := "Unit1.EmNodes".unitRecipe.unitRecipe.electrodWidth;
       "Unit1.MotionNodes".PLCToMotion.Parameter.MeasureIMain.Tab.TabToEdge := "Unit1.EmNodes".unitRecipe.unitRecipe.electrodTabToEdge;
       "Unit1.MotionNodes".PLCToMotion.Parameter.MeasureIMain.Tab.CutDistances := "Unit1.EmNodes".unitRecipe.unitRecipe.TabSensorToCutterDistance;
       "Unit1.MotionNodes".PLCToMotion.Parameter.MeasureIMain.Tab.CutDistancesOffset := 0.0;
   END_IF;
END_REGION

REGION Network 85: Parameter MeasureIMain Joint
   RUNG wire#powerrail
      Contact( #TRUE )
      Move(in := 0.0, out1 => "Unit1.MotionNodes".PLCToMotion.Parameter.MeasureIMain.Joint.JointFilterDistance)
      Move(in := 0.0, out1 => "Unit1.MotionNodes".PLCToMotion.Parameter.MeasureIMain.Joint.JointSensorToCutDistance)
   END_RUNG
   // the same network as SCL:
   IF #TRUE THEN
       "Unit1.MotionNodes".PLCToMotion.Parameter.MeasureIMain.Joint.JointFilterDistance := 0.0;
       "Unit1.MotionNodes".PLCToMotion.Parameter.MeasureIMain.Joint.JointSensorToCutDistance := 0.0;
   END_IF;
END_REGION

REGION Network 86: Parameter MeasureIMain Cell
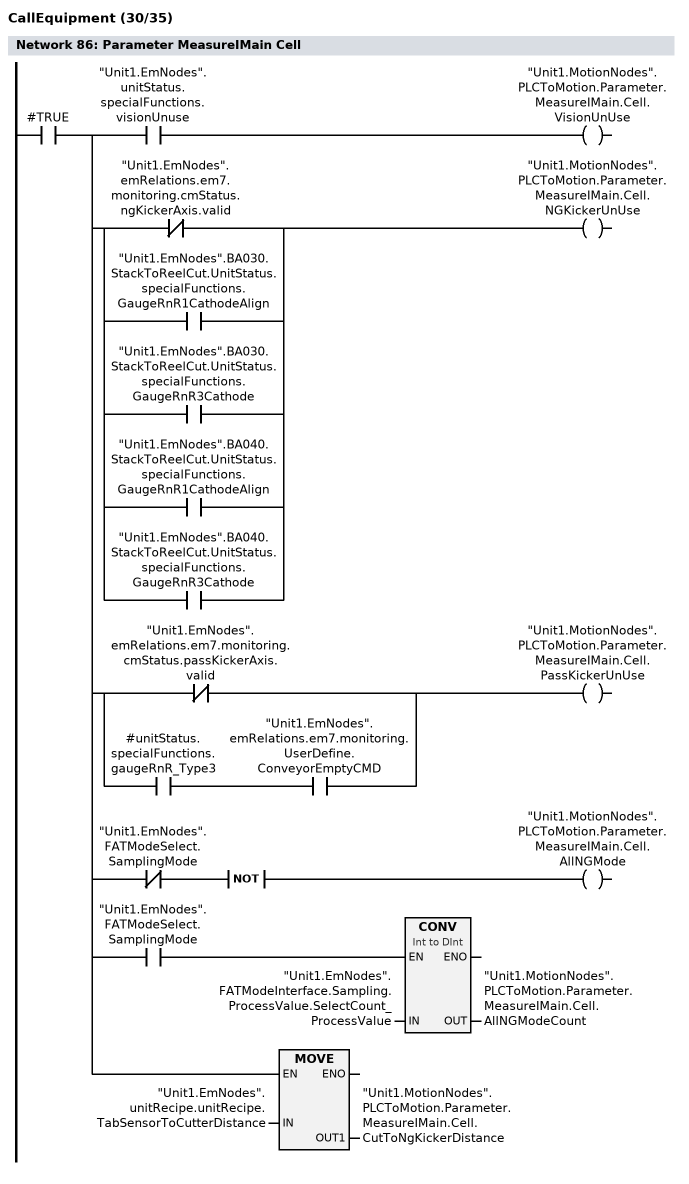
   RUNG wire#powerrail
      Contact( #TRUE )
      wire#w1
      Contact( "Unit1.EmNodes".unitStatus.specialFunctions.visionUnuse )
      Coil( "Unit1.MotionNodes".PLCToMotion.Parameter.MeasureIMain.Cell.VisionUnUse )
   END_RUNG
   RUNG wire#w1
      I_Contact( "Unit1.EmNodes".emRelations.em7.monitoring.cmStatus.ngKickerAxis.valid )
      wire#w2
      Coil( "Unit1.MotionNodes".PLCToMotion.Parameter.MeasureIMain.Cell.NGKickerUnUse )
   END_RUNG
   RUNG wire#w1
      Contact( "Unit1.EmNodes".BA030.StackToReelCut.UnitStatus.specialFunctions.GaugeRnR1CathodeAlign )
   END_RUNG wire#w2
   RUNG wire#w1
      Contact( "Unit1.EmNodes".BA030.StackToReelCut.UnitStatus.specialFunctions.GaugeRnR3Cathode )
   END_RUNG wire#w2
   RUNG wire#w1
      Contact( "Unit1.EmNodes".BA040.StackToReelCut.UnitStatus.specialFunctions.GaugeRnR1CathodeAlign )
   END_RUNG wire#w2
   RUNG wire#w1
      Contact( "Unit1.EmNodes".BA040.StackToReelCut.UnitStatus.specialFunctions.GaugeRnR3Cathode )
   END_RUNG wire#w2
   RUNG wire#w1
      I_Contact( "Unit1.EmNodes".emRelations.em7.monitoring.cmStatus.passKickerAxis.valid )
      wire#w3
      Coil( "Unit1.MotionNodes".PLCToMotion.Parameter.MeasureIMain.Cell.PassKickerUnUse )
   END_RUNG
   RUNG wire#w1
      Contact( #unitStatus.specialFunctions.gaugeRnR_Type3 )
      Contact( "Unit1.EmNodes".emRelations.em7.monitoring.UserDefine.ConveyorEmptyCMD )
   END_RUNG wire#w3
   RUNG wire#w1
      I_Contact( "Unit1.EmNodes".FATModeSelect.SamplingMode )
      Not()
      Coil( "Unit1.MotionNodes".PLCToMotion.Parameter.MeasureIMain.Cell.AllNGMode )
   END_RUNG
   RUNG wire#w1
      Contact( "Unit1.EmNodes".FATModeSelect.SamplingMode )
      { S7_Templates := "[SrcType := Int, DestType := DInt]" } Convert(in := "Unit1.EmNodes".FATModeInterface.Sampling.ProcessValue.SelectCount_ProcessValue, out => "Unit1.MotionNodes".PLCToMotion.Parameter.MeasureIMain.Cell.AllNGModeCount)
   END_RUNG
   RUNG wire#w1
      Move(in := "Unit1.EmNodes".unitRecipe.unitRecipe.TabSensorToCutterDistance, out1 => "Unit1.MotionNodes".PLCToMotion.Parameter.MeasureIMain.Cell.CutToNgKickerDistance)
   END_RUNG
   // the same network as SCL:
   "Unit1.MotionNodes".PLCToMotion.Parameter.MeasureIMain.Cell.VisionUnUse := #TRUE AND "Unit1.EmNodes".unitStatus.specialFunctions.visionUnuse;
   "Unit1.MotionNodes".PLCToMotion.Parameter.MeasureIMain.Cell.NGKickerUnUse := #TRUE AND (NOT "Unit1.EmNodes".emRelations.em7.monitoring.cmStatus.ngKickerAxis.valid OR "Unit1.EmNodes".BA030.StackToReelCut.UnitStatus.specialFunctions.GaugeRnR1CathodeAlign OR "Unit1.EmNodes".BA030.StackToReelCut.UnitStatus.specialFunctions.GaugeRnR3Cathode OR "Unit1.EmNodes".BA040.StackToReelCut.UnitStatus.specialFunctions.GaugeRnR1CathodeAlign OR "Unit1.EmNodes".BA040.StackToReelCut.UnitStatus.specialFunctions.GaugeRnR3Cathode);
   "Unit1.MotionNodes".PLCToMotion.Parameter.MeasureIMain.Cell.PassKickerUnUse := #TRUE AND (NOT "Unit1.EmNodes".emRelations.em7.monitoring.cmStatus.passKickerAxis.valid OR (#unitStatus.specialFunctions.gaugeRnR_Type3 AND "Unit1.EmNodes".emRelations.em7.monitoring.UserDefine.ConveyorEmptyCMD));
   "Unit1.MotionNodes".PLCToMotion.Parameter.MeasureIMain.Cell.AllNGMode := NOT (#TRUE AND NOT "Unit1.EmNodes".FATModeSelect.SamplingMode);
   IF #TRUE AND "Unit1.EmNodes".FATModeSelect.SamplingMode THEN
       "Unit1.MotionNodes".PLCToMotion.Parameter.MeasureIMain.Cell.AllNGModeCount := INT_TO_DINT("Unit1.EmNodes".FATModeInterface.Sampling.ProcessValue.SelectCount_ProcessValue);
   END_IF;
   IF #TRUE THEN
       "Unit1.MotionNodes".PLCToMotion.Parameter.MeasureIMain.Cell.CutToNgKickerDistance := "Unit1.EmNodes".unitRecipe.unitRecipe.TabSensorToCutterDistance;
   END_IF;
END_REGION

REGION Network 87: Parameter MeasureIMain Vision
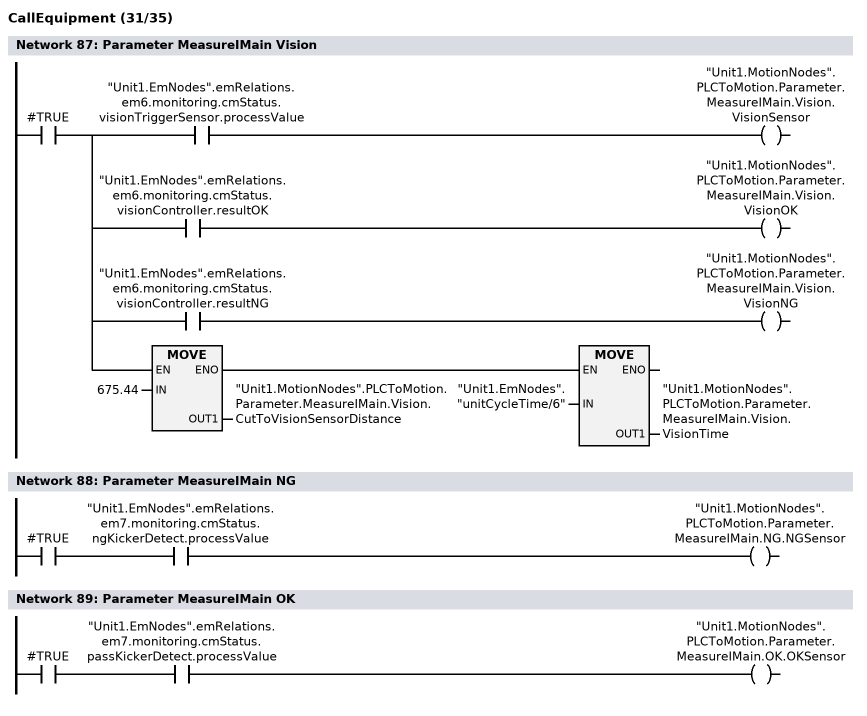
   RUNG wire#powerrail
      Contact( #TRUE )
      wire#w1
      Contact( "Unit1.EmNodes".emRelations.em6.monitoring.cmStatus.visionTriggerSensor.processValue )
      Coil( "Unit1.MotionNodes".PLCToMotion.Parameter.MeasureIMain.Vision.VisionSensor )
   END_RUNG
   RUNG wire#w1
      Contact( "Unit1.EmNodes".emRelations.em6.monitoring.cmStatus.visionController.resultOK )
      Coil( "Unit1.MotionNodes".PLCToMotion.Parameter.MeasureIMain.Vision.VisionOK )
   END_RUNG
   RUNG wire#w1
      Contact( "Unit1.EmNodes".emRelations.em6.monitoring.cmStatus.visionController.resultNG )
      Coil( "Unit1.MotionNodes".PLCToMotion.Parameter.MeasureIMain.Vision.VisionNG )
   END_RUNG
   RUNG wire#w1
      Move(in := 675.44, out1 => "Unit1.MotionNodes".PLCToMotion.Parameter.MeasureIMain.Vision.CutToVisionSensorDistance)
      Move(in := "Unit1.EmNodes"."unitCycleTime/6", out1 => "Unit1.MotionNodes".PLCToMotion.Parameter.MeasureIMain.Vision.VisionTime)
   END_RUNG
   // the same network as SCL:
   "Unit1.MotionNodes".PLCToMotion.Parameter.MeasureIMain.Vision.VisionSensor := #TRUE AND "Unit1.EmNodes".emRelations.em6.monitoring.cmStatus.visionTriggerSensor.processValue;
   "Unit1.MotionNodes".PLCToMotion.Parameter.MeasureIMain.Vision.VisionOK := #TRUE AND "Unit1.EmNodes".emRelations.em6.monitoring.cmStatus.visionController.resultOK;
   "Unit1.MotionNodes".PLCToMotion.Parameter.MeasureIMain.Vision.VisionNG := #TRUE AND "Unit1.EmNodes".emRelations.em6.monitoring.cmStatus.visionController.resultNG;
   IF #TRUE THEN
       "Unit1.MotionNodes".PLCToMotion.Parameter.MeasureIMain.Vision.CutToVisionSensorDistance := 675.44;
       "Unit1.MotionNodes".PLCToMotion.Parameter.MeasureIMain.Vision.VisionTime := "Unit1.EmNodes"."unitCycleTime/6";
   END_IF;
END_REGION

REGION Network 88: Parameter MeasureIMain NG
   RUNG wire#powerrail
      Contact( #TRUE )
      Contact( "Unit1.EmNodes".emRelations.em7.monitoring.cmStatus.ngKickerDetect.processValue )
      Coil( "Unit1.MotionNodes".PLCToMotion.Parameter.MeasureIMain.NG.NGSensor )
   END_RUNG
   // the same network as SCL:
   "Unit1.MotionNodes".PLCToMotion.Parameter.MeasureIMain.NG.NGSensor := #TRUE AND "Unit1.EmNodes".emRelations.em7.monitoring.cmStatus.ngKickerDetect.processValue;
END_REGION

REGION Network 89: Parameter MeasureIMain OK
   RUNG wire#powerrail
      Contact( #TRUE )
      Contact( "Unit1.EmNodes".emRelations.em7.monitoring.cmStatus.passKickerDetect.processValue )
      Coil( "Unit1.MotionNodes".PLCToMotion.Parameter.MeasureIMain.OK.OKSensor )
   END_RUNG
   // the same network as SCL:
   "Unit1.MotionNodes".PLCToMotion.Parameter.MeasureIMain.OK.OKSensor := #TRUE AND "Unit1.EmNodes".emRelations.em7.monitoring.cmStatus.passKickerDetect.processValue;
END_REGION

REGION Network 90: ******************** Feedback to Unit ********************
END_REGION

REGION Network 91: Determine StateComplete (SC) in Mode Production
   // Conditions for the Equipment Modules "stateComplete" feedback to the unit. This feedback is given when the task in for the respective state is complete.
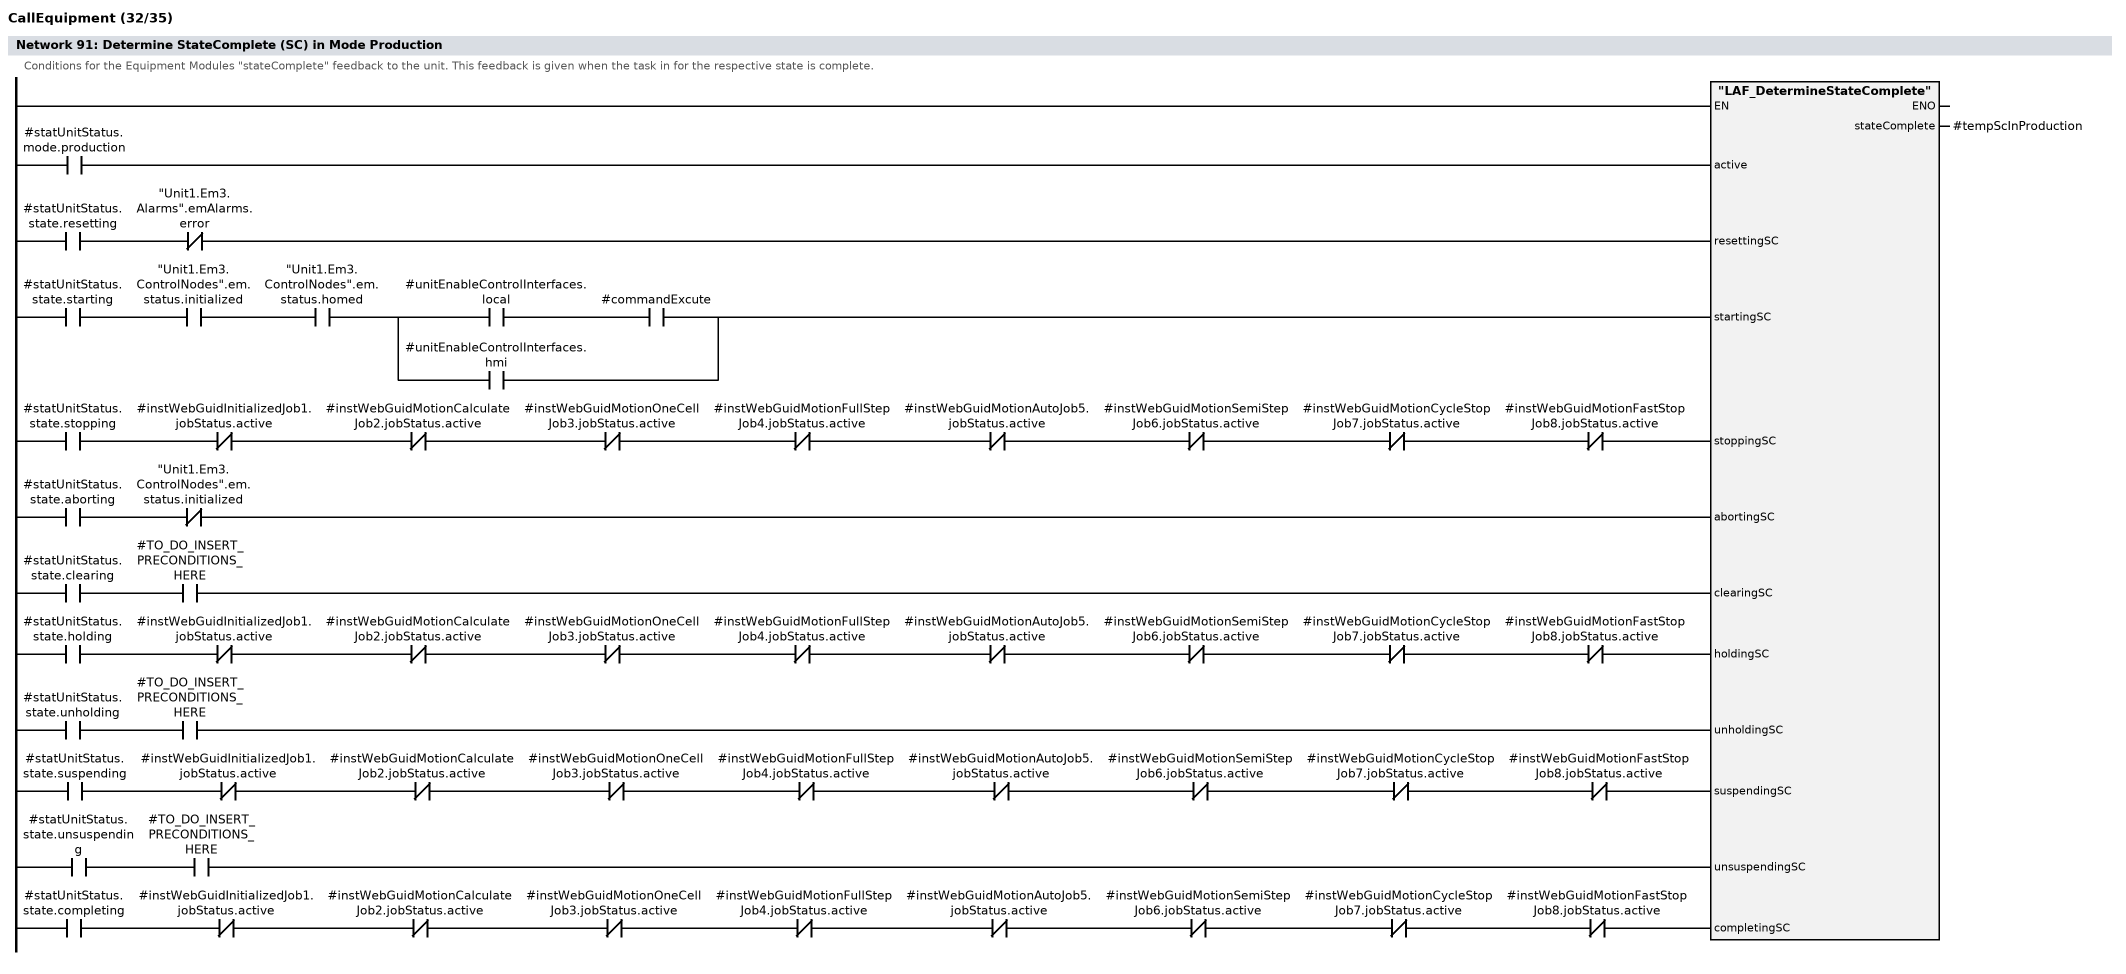
   RUNG wire#powerrail
      "LAF_DetermineStateComplete"(active := wire#w1, resettingSC := wire#w2, startingSC := wire#w4, stoppingSC := wire#w5, abortingSC := wire#w6, clearingSC := wire#w7, holdingSC := wire#w8, unholdingSC := wire#w9, suspendingSC := wire#w10, unsuspendingSC := wire#w11, completingSC := wire#w12, stateComplete => #tempScInProduction)
   END_RUNG
   RUNG wire#powerrail
      Contact( #statUnitStatus.mode.production )
   END_RUNG wire#w1
   RUNG wire#powerrail
      Contact( #statUnitStatus.state.resetting )
      I_Contact( "Unit1.Em3.Alarms".emAlarms.error )
   END_RUNG wire#w2
   RUNG wire#powerrail
      Contact( #statUnitStatus.state.starting )
      Contact( "Unit1.Em3.ControlNodes".em.status.initialized )
      Contact( "Unit1.Em3.ControlNodes".em.status.homed )
      wire#w3
      Contact( #unitEnableControlInterfaces.local )
      Contact( #commandExcute )
   END_RUNG wire#w4
   RUNG wire#w3
      Contact( #unitEnableControlInterfaces.hmi )
   END_RUNG wire#w4
   RUNG wire#powerrail
      Contact( #statUnitStatus.state.stopping )
      I_Contact( #instWebGuidInitializedJob1.jobStatus.active )
      I_Contact( #instWebGuidMotionCalculateJob2.jobStatus.active )
      I_Contact( #instWebGuidMotionOneCellJob3.jobStatus.active )
      I_Contact( #instWebGuidMotionFullStepJob4.jobStatus.active )
      I_Contact( #instWebGuidMotionAutoJob5.jobStatus.active )
      I_Contact( #instWebGuidMotionSemiStepJob6.jobStatus.active )
      I_Contact( #instWebGuidMotionCycleStopJob7.jobStatus.active )
      I_Contact( #instWebGuidMotionFastStopJob8.jobStatus.active )
   END_RUNG wire#w5
   RUNG wire#powerrail
      Contact( #statUnitStatus.state.aborting )
      I_Contact( "Unit1.Em3.ControlNodes".em.status.initialized )
   END_RUNG wire#w6
   RUNG wire#powerrail
      Contact( #statUnitStatus.state.clearing )
      Contact( #TO_DO_INSERT_PRECONDITIONS_HERE )
   END_RUNG wire#w7
   RUNG wire#powerrail
      Contact( #statUnitStatus.state.holding )
      I_Contact( #instWebGuidInitializedJob1.jobStatus.active )
      I_Contact( #instWebGuidMotionCalculateJob2.jobStatus.active )
      I_Contact( #instWebGuidMotionOneCellJob3.jobStatus.active )
      I_Contact( #instWebGuidMotionFullStepJob4.jobStatus.active )
      I_Contact( #instWebGuidMotionAutoJob5.jobStatus.active )
      I_Contact( #instWebGuidMotionSemiStepJob6.jobStatus.active )
      I_Contact( #instWebGuidMotionCycleStopJob7.jobStatus.active )
      I_Contact( #instWebGuidMotionFastStopJob8.jobStatus.active )
   END_RUNG wire#w8
   RUNG wire#powerrail
      Contact( #statUnitStatus.state.unholding )
      Contact( #TO_DO_INSERT_PRECONDITIONS_HERE )
   END_RUNG wire#w9
   RUNG wire#powerrail
      Contact( #statUnitStatus.state.suspending )
      I_Contact( #instWebGuidInitializedJob1.jobStatus.active )
      I_Contact( #instWebGuidMotionCalculateJob2.jobStatus.active )
      I_Contact( #instWebGuidMotionOneCellJob3.jobStatus.active )
      I_Contact( #instWebGuidMotionFullStepJob4.jobStatus.active )
      I_Contact( #instWebGuidMotionAutoJob5.jobStatus.active )
      I_Contact( #instWebGuidMotionSemiStepJob6.jobStatus.active )
      I_Contact( #instWebGuidMotionCycleStopJob7.jobStatus.active )
      I_Contact( #instWebGuidMotionFastStopJob8.jobStatus.active )
   END_RUNG wire#w10
   RUNG wire#powerrail
      Contact( #statUnitStatus.state.unsuspending )
      Contact( #TO_DO_INSERT_PRECONDITIONS_HERE )
   END_RUNG wire#w11
   RUNG wire#powerrail
      Contact( #statUnitStatus.state.completing )
      I_Contact( #instWebGuidInitializedJob1.jobStatus.active )
      I_Contact( #instWebGuidMotionCalculateJob2.jobStatus.active )
      I_Contact( #instWebGuidMotionOneCellJob3.jobStatus.active )
      I_Contact( #instWebGuidMotionFullStepJob4.jobStatus.active )
      I_Contact( #instWebGuidMotionAutoJob5.jobStatus.active )
      I_Contact( #instWebGuidMotionSemiStepJob6.jobStatus.active )
      I_Contact( #instWebGuidMotionCycleStopJob7.jobStatus.active )
      I_Contact( #instWebGuidMotionFastStopJob8.jobStatus.active )
   END_RUNG wire#w12
   // the same network as SCL:
   "LAF_DetermineStateComplete"(active := #statUnitStatus.mode.production,
                           resettingSC := #statUnitStatus.state.resetting AND NOT "Unit1.Em3.Alarms".emAlarms.error,
                           startingSC := #statUnitStatus.state.starting AND "Unit1.Em3.ControlNodes".em.status.initialized AND "Unit1.Em3.ControlNodes".em.status.homed AND ((#unitEnableControlInterfaces.local AND #commandExcute) OR #unitEnableControlInterfaces.hmi),
                           stoppingSC := #statUnitStatus.state.stopping AND NOT #instWebGuidInitializedJob1.jobStatus.active AND NOT #instWebGuidMotionCalculateJob2.jobStatus.active AND NOT #instWebGuidMotionOneCellJob3.jobStatus.active AND NOT #instWebGuidMotionFullStepJob4.jobStatus.active AND NOT #instWebGuidMotionAutoJob5.jobStatus.active AND NOT #instWebGuidMotionSemiStepJob6.jobStatus.active AND NOT #instWebGuidMotionCycleStopJob7.jobStatus.active AND NOT #instWebGuidMotionFastStopJob8.jobStatus.active,
                           abortingSC := #statUnitStatus.state.aborting AND NOT "Unit1.Em3.ControlNodes".em.status.initialized,
                           clearingSC := #statUnitStatus.state.clearing AND #TO_DO_INSERT_PRECONDITIONS_HERE,
                           holdingSC := #statUnitStatus.state.holding AND NOT #instWebGuidInitializedJob1.jobStatus.active AND NOT #instWebGuidMotionCalculateJob2.jobStatus.active AND NOT #instWebGuidMotionOneCellJob3.jobStatus.active AND NOT #instWebGuidMotionFullStepJob4.jobStatus.active AND NOT #instWebGuidMotionAutoJob5.jobStatus.active AND NOT #instWebGuidMotionSemiStepJob6.jobStatus.active AND NOT #instWebGuidMotionCycleStopJob7.jobStatus.active AND NOT #instWebGuidMotionFastStopJob8.jobStatus.active,
                           unholdingSC := #statUnitStatus.state.unholding AND #TO_DO_INSERT_PRECONDITIONS_HERE,
                           suspendingSC := #statUnitStatus.state.suspending AND NOT #instWebGuidInitializedJob1.jobStatus.active AND NOT #instWebGuidMotionCalculateJob2.jobStatus.active AND NOT #instWebGuidMotionOneCellJob3.jobStatus.active AND NOT #instWebGuidMotionFullStepJob4.jobStatus.active AND NOT #instWebGuidMotionAutoJob5.jobStatus.active AND NOT #instWebGuidMotionSemiStepJob6.jobStatus.active AND NOT #instWebGuidMotionCycleStopJob7.jobStatus.active AND NOT #instWebGuidMotionFastStopJob8.jobStatus.active,
                           unsuspendingSC := #statUnitStatus.state.unsuspending AND #TO_DO_INSERT_PRECONDITIONS_HERE,
                           completingSC := #statUnitStatus.state.completing AND NOT #instWebGuidInitializedJob1.jobStatus.active AND NOT #instWebGuidMotionCalculateJob2.jobStatus.active AND NOT #instWebGuidMotionOneCellJob3.jobStatus.active AND NOT #instWebGuidMotionFullStepJob4.jobStatus.active AND NOT #instWebGuidMotionAutoJob5.jobStatus.active AND NOT #instWebGuidMotionSemiStepJob6.jobStatus.active AND NOT #instWebGuidMotionCycleStopJob7.jobStatus.active AND NOT #instWebGuidMotionFastStopJob8.jobStatus.active,
                           stateComplete => #tempScInProduction);
END_REGION

REGION Network 92: Determine StateComplete (SC) in Mode Maintenance/Manual
   // Conditions for the Equipment Modules "stateComplete" feedback to the unit. This feedback is given when the task in for the respective state is complete.
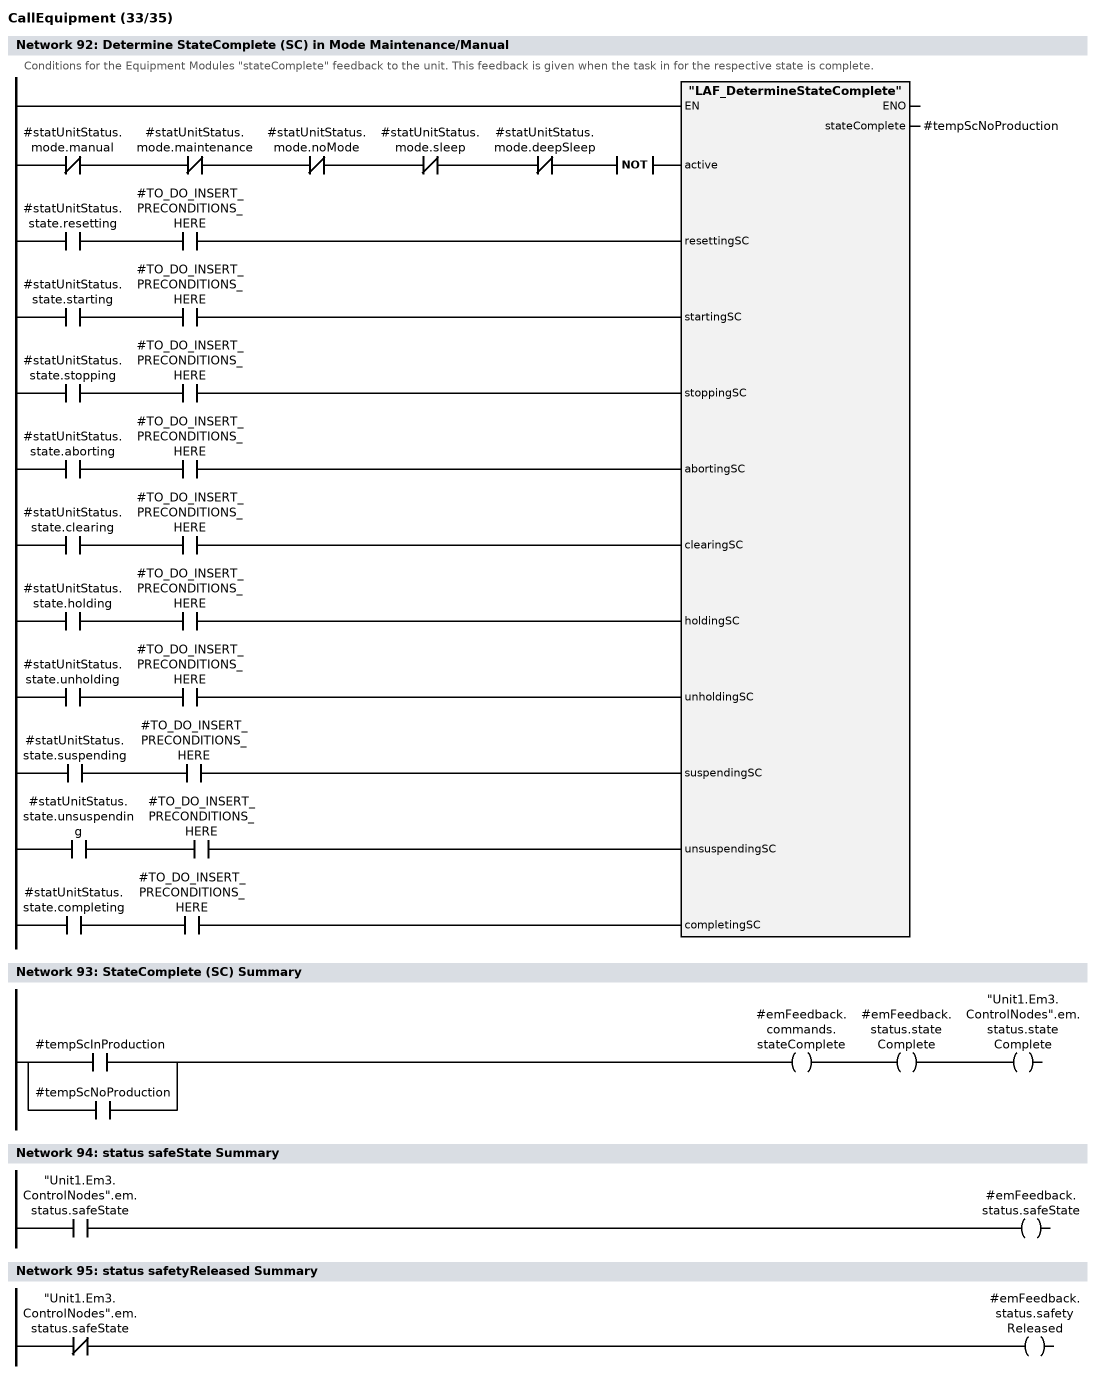
   RUNG wire#powerrail
      "LAF_DetermineStateComplete"(active := wire#w1, resettingSC := wire#w2, startingSC := wire#w3, stoppingSC := wire#w4, abortingSC := wire#w5, clearingSC := wire#w6, holdingSC := wire#w7, unholdingSC := wire#w8, suspendingSC := wire#w9, unsuspendingSC := wire#w10, completingSC := wire#w11, stateComplete => #tempScNoProduction)
   END_RUNG
   RUNG wire#powerrail
      I_Contact( #statUnitStatus.mode.manual )
      I_Contact( #statUnitStatus.mode.maintenance )
      I_Contact( #statUnitStatus.mode.noMode )
      I_Contact( #statUnitStatus.mode.sleep )
      I_Contact( #statUnitStatus.mode.deepSleep )
      Not()
   END_RUNG wire#w1
   RUNG wire#powerrail
      Contact( #statUnitStatus.state.resetting )
      Contact( #TO_DO_INSERT_PRECONDITIONS_HERE )
   END_RUNG wire#w2
   RUNG wire#powerrail
      Contact( #statUnitStatus.state.starting )
      Contact( #TO_DO_INSERT_PRECONDITIONS_HERE )
   END_RUNG wire#w3
   RUNG wire#powerrail
      Contact( #statUnitStatus.state.stopping )
      Contact( #TO_DO_INSERT_PRECONDITIONS_HERE )
   END_RUNG wire#w4
   RUNG wire#powerrail
      Contact( #statUnitStatus.state.aborting )
      Contact( #TO_DO_INSERT_PRECONDITIONS_HERE )
   END_RUNG wire#w5
   RUNG wire#powerrail
      Contact( #statUnitStatus.state.clearing )
      Contact( #TO_DO_INSERT_PRECONDITIONS_HERE )
   END_RUNG wire#w6
   RUNG wire#powerrail
      Contact( #statUnitStatus.state.holding )
      Contact( #TO_DO_INSERT_PRECONDITIONS_HERE )
   END_RUNG wire#w7
   RUNG wire#powerrail
      Contact( #statUnitStatus.state.unholding )
      Contact( #TO_DO_INSERT_PRECONDITIONS_HERE )
   END_RUNG wire#w8
   RUNG wire#powerrail
      Contact( #statUnitStatus.state.suspending )
      Contact( #TO_DO_INSERT_PRECONDITIONS_HERE )
   END_RUNG wire#w9
   RUNG wire#powerrail
      Contact( #statUnitStatus.state.unsuspending )
      Contact( #TO_DO_INSERT_PRECONDITIONS_HERE )
   END_RUNG wire#w10
   RUNG wire#powerrail
      Contact( #statUnitStatus.state.completing )
      Contact( #TO_DO_INSERT_PRECONDITIONS_HERE )
   END_RUNG wire#w11
   // the same network as SCL:
   "LAF_DetermineStateComplete"(active := NOT (NOT #statUnitStatus.mode.manual AND NOT #statUnitStatus.mode.maintenance AND NOT #statUnitStatus.mode.noMode AND NOT #statUnitStatus.mode.sleep AND NOT #statUnitStatus.mode.deepSleep),
                           resettingSC := #statUnitStatus.state.resetting AND #TO_DO_INSERT_PRECONDITIONS_HERE,
                           startingSC := #statUnitStatus.state.starting AND #TO_DO_INSERT_PRECONDITIONS_HERE,
                           stoppingSC := #statUnitStatus.state.stopping AND #TO_DO_INSERT_PRECONDITIONS_HERE,
                           abortingSC := #statUnitStatus.state.aborting AND #TO_DO_INSERT_PRECONDITIONS_HERE,
                           clearingSC := #statUnitStatus.state.clearing AND #TO_DO_INSERT_PRECONDITIONS_HERE,
                           holdingSC := #statUnitStatus.state.holding AND #TO_DO_INSERT_PRECONDITIONS_HERE,
                           unholdingSC := #statUnitStatus.state.unholding AND #TO_DO_INSERT_PRECONDITIONS_HERE,
                           suspendingSC := #statUnitStatus.state.suspending AND #TO_DO_INSERT_PRECONDITIONS_HERE,
                           unsuspendingSC := #statUnitStatus.state.unsuspending AND #TO_DO_INSERT_PRECONDITIONS_HERE,
                           completingSC := #statUnitStatus.state.completing AND #TO_DO_INSERT_PRECONDITIONS_HERE,
                           stateComplete => #tempScNoProduction);
END_REGION

REGION Network 93: StateComplete (SC) Summary
   RUNG wire#powerrail
      Contact( #tempScInProduction )
      wire#w1
      Coil( #emFeedback.commands.stateComplete )
      Coil( #emFeedback.status.stateComplete )
      Coil( "Unit1.Em3.ControlNodes".em.status.stateComplete )
   END_RUNG
   RUNG wire#powerrail
      Contact( #tempScNoProduction )
   END_RUNG wire#w1
   // the same network as SCL:
   #emFeedback.commands.stateComplete := #tempScInProduction OR #tempScNoProduction;
   #emFeedback.status.stateComplete := #emFeedback.commands.stateComplete;
   "Unit1.Em3.ControlNodes".em.status.stateComplete := #emFeedback.commands.stateComplete;
END_REGION

REGION Network 94: status safeState Summary
   RUNG wire#powerrail
      Contact( "Unit1.Em3.ControlNodes".em.status.safeState )
      Coil( #emFeedback.status.safeState )
   END_RUNG
   // the same network as SCL:
   #emFeedback.status.safeState := "Unit1.Em3.ControlNodes".em.status.safeState;
END_REGION

REGION Network 95: status safetyReleased Summary
   RUNG wire#powerrail
      I_Contact( "Unit1.Em3.ControlNodes".em.status.safeState )
      Coil( #emFeedback.status.safetyReleased )
   END_RUNG
   // the same network as SCL:
   #emFeedback.status.safetyReleased := NOT "Unit1.Em3.ControlNodes".em.status.safeState;
END_REGION

REGION Network 96: ******************** Alarms ********************
END_REGION

REGION Network 97: Collet Alarms
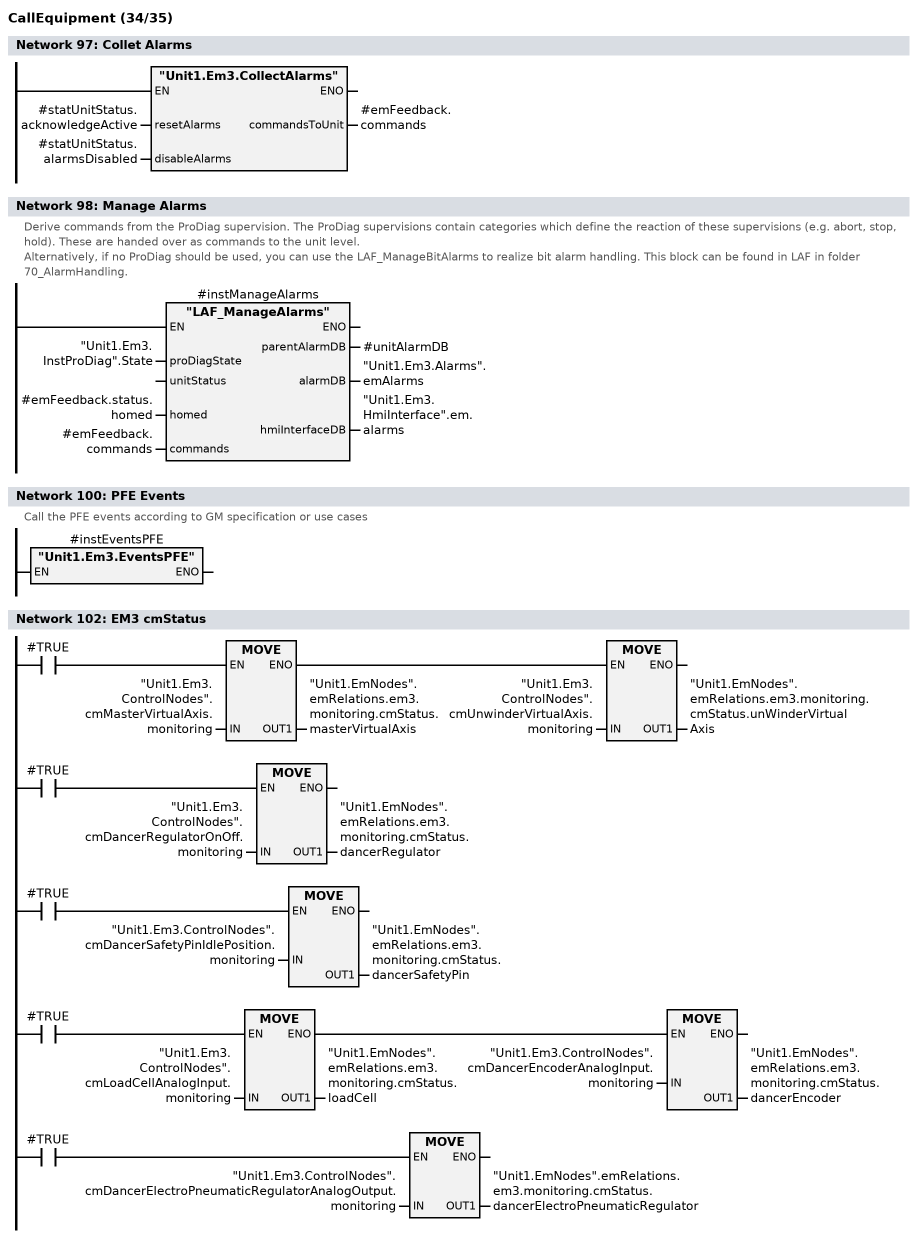
   RUNG wire#powerrail
      "Unit1.Em3.CollectAlarms"(resetAlarms := #statUnitStatus.acknowledgeActive, disableAlarms := #statUnitStatus.alarmsDisabled, commandsToUnit => #emFeedback.commands)
   END_RUNG
   // the same network as SCL:
   "Unit1.Em3.CollectAlarms"(resetAlarms := #statUnitStatus.acknowledgeActive,
                           disableAlarms := #statUnitStatus.alarmsDisabled,
                           commandsToUnit => #emFeedback.commands);
END_REGION

REGION Network 98: Manage Alarms
   // Derive commands from the ProDiag supervision. The ProDiag supervisions contain categories which define the reaction of these supervisions (e.g. abort, stop, hold). These are handed over as commands to the unit level.
   // Alternatively, if no ProDiag should be used, you can use the LAF_ManageBitAlarms to realize bit alarm handling. This block can be found in LAF in folder 70_AlarmHandling.
   RUNG wire#powerrail
      #instManageAlarms(proDiagState := "Unit1.Em3.InstProDiag".State, unitStatus :=, homed := #emFeedback.status.homed, commands := #emFeedback.commands, parentAlarmDB => #unitAlarmDB, alarmDB => "Unit1.Em3.Alarms".emAlarms, hmiInterfaceDB => "Unit1.Em3.HmiInterface".em.alarms)
   END_RUNG
   // the same network as SCL:
   #instManageAlarms(proDiagState := "Unit1.Em3.InstProDiag".State,   // "LAF_ManageAlarms"
                     homed := #emFeedback.status.homed,
                     commands := #emFeedback.commands,
                     parentAlarmDB => #unitAlarmDB,
                     alarmDB => "Unit1.Em3.Alarms".emAlarms,
                     hmiInterfaceDB => "Unit1.Em3.HmiInterface".em.alarms);
END_REGION

REGION Network 99: ******************** PFE Events ********************
END_REGION

REGION Network 100: PFE Events
   // Call the PFE events according to GM specification or use cases
   RUNG wire#powerrail
      #instEventsPFE()
   END_RUNG
   // the same network as SCL:
   #instEventsPFE();   // "Unit1.Em3.EventsPFE"
END_REGION

REGION Network 101: ******************** EM Relations Output ********************
END_REGION

REGION Network 102: EM3 cmStatus
   RUNG wire#powerrail
      Contact( #TRUE )
      Move(in := "Unit1.Em3.ControlNodes".cmMasterVirtualAxis.monitoring, out1 => "Unit1.EmNodes".emRelations.em3.monitoring.cmStatus.masterVirtualAxis)
      Move(in := "Unit1.Em3.ControlNodes".cmUnwinderVirtualAxis.monitoring, out1 => "Unit1.EmNodes".emRelations.em3.monitoring.cmStatus.unWinderVirtualAxis)
   END_RUNG
   RUNG wire#powerrail
      Contact( #TRUE )
      Move(in := "Unit1.Em3.ControlNodes".cmDancerRegulatorOnOff.monitoring, out1 => "Unit1.EmNodes".emRelations.em3.monitoring.cmStatus.dancerRegulator)
   END_RUNG
   RUNG wire#powerrail
      Contact( #TRUE )
      Move(in := "Unit1.Em3.ControlNodes".cmDancerSafetyPinIdlePosition.monitoring, out1 => "Unit1.EmNodes".emRelations.em3.monitoring.cmStatus.dancerSafetyPin)
   END_RUNG
   RUNG wire#powerrail
      Contact( #TRUE )
      Move(in := "Unit1.Em3.ControlNodes".cmLoadCellAnalogInput.monitoring, out1 => "Unit1.EmNodes".emRelations.em3.monitoring.cmStatus.loadCell)
      Move(in := "Unit1.Em3.ControlNodes".cmDancerEncoderAnalogInput.monitoring, out1 => "Unit1.EmNodes".emRelations.em3.monitoring.cmStatus.dancerEncoder)
   END_RUNG
   RUNG wire#powerrail
      Contact( #TRUE )
      Move(in := "Unit1.Em3.ControlNodes".cmDancerElectroPneumaticRegulatorAnalogOutput.monitoring, out1 => "Unit1.EmNodes".emRelations.em3.monitoring.cmStatus.dancerElectroPneumaticRegulator)
   END_RUNG
   // the same network as SCL:
   IF #TRUE THEN
       "Unit1.EmNodes".emRelations.em3.monitoring.cmStatus.masterVirtualAxis := "Unit1.Em3.ControlNodes".cmMasterVirtualAxis.monitoring;
       "Unit1.EmNodes".emRelations.em3.monitoring.cmStatus.unWinderVirtualAxis := "Unit1.Em3.ControlNodes".cmUnwinderVirtualAxis.monitoring;
       "Unit1.EmNodes".emRelations.em3.monitoring.cmStatus.dancerRegulator := "Unit1.Em3.ControlNodes".cmDancerRegulatorOnOff.monitoring;
       "Unit1.EmNodes".emRelations.em3.monitoring.cmStatus.dancerSafetyPin := "Unit1.Em3.ControlNodes".cmDancerSafetyPinIdlePosition.monitoring;
       "Unit1.EmNodes".emRelations.em3.monitoring.cmStatus.loadCell := "Unit1.Em3.ControlNodes".cmLoadCellAnalogInput.monitoring;
       "Unit1.EmNodes".emRelations.em3.monitoring.cmStatus.dancerEncoder := "Unit1.Em3.ControlNodes".cmDancerEncoderAnalogInput.monitoring;
       "Unit1.EmNodes".emRelations.em3.monitoring.cmStatus.dancerElectroPneumaticRegulator := "Unit1.Em3.ControlNodes".cmDancerElectroPneumaticRegulatorAnalogOutput.monitoring;
   END_IF;
END_REGION

REGION Network 103: EM3 UserDefine
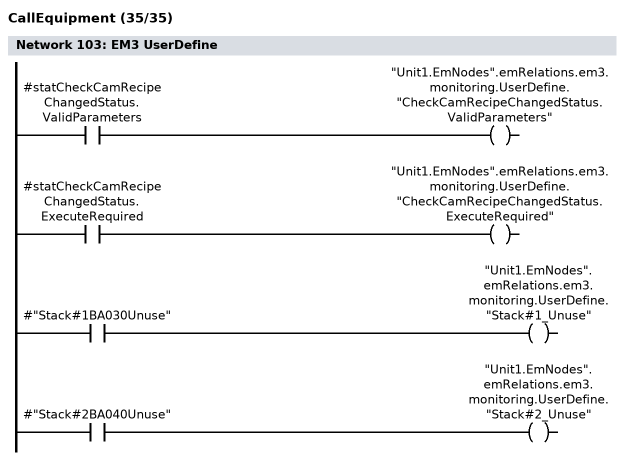
   RUNG wire#powerrail
      Contact( #statCheckCamRecipeChangedStatus.ValidParameters )
      Coil( "Unit1.EmNodes".emRelations.em3.monitoring.UserDefine."CheckCamRecipeChangedStatus.ValidParameters" )
   END_RUNG
   RUNG wire#powerrail
      Contact( #statCheckCamRecipeChangedStatus.ExecuteRequired )
      Coil( "Unit1.EmNodes".emRelations.em3.monitoring.UserDefine."CheckCamRecipeChangedStatus.ExecuteRequired" )
   END_RUNG
   RUNG wire#powerrail
      Contact( #"Stack#1BA030Unuse" )
      Coil( "Unit1.EmNodes".emRelations.em3.monitoring.UserDefine."Stack#1_Unuse" )
   END_RUNG
   RUNG wire#powerrail
      Contact( #"Stack#2BA040Unuse" )
      Coil( "Unit1.EmNodes".emRelations.em3.monitoring.UserDefine."Stack#2_Unuse" )
   END_RUNG
   // the same network as SCL:
   "Unit1.EmNodes".emRelations.em3.monitoring.UserDefine."CheckCamRecipeChangedStatus.ValidParameters" := #statCheckCamRecipeChangedStatus.ValidParameters;
   "Unit1.EmNodes".emRelations.em3.monitoring.UserDefine."CheckCamRecipeChangedStatus.ExecuteRequired" := #statCheckCamRecipeChangedStatus.ExecuteRequired;
   "Unit1.EmNodes".emRelations.em3.monitoring.UserDefine."Stack#1_Unuse" := #"Stack#1BA030Unuse";
   "Unit1.EmNodes".emRelations.em3.monitoring.UserDefine."Stack#2_Unuse" := #"Stack#2BA040Unuse";
END_REGION
END_FUNCTION_BLOCK
